		6:	IF (NOT(T_Station_Work.THWWorkStation.TAxisZ.T_CtrleSingle.xReset) AND (T_Station_Work.THWWorkStation.TAxisZ.T_CtrleSingle.xDone OR
			     T_Station_Work.THWWorkStation.TAxisZ.T_CtrleSingle.xErr)) OR
			    (NOT(T_Station_Work.THWWorkStation.TAxisS.T_CtrleSingle.xReset) AND (T_Station_Work.THWWorkStation.TAxisS.T_CtrleSingle.xDone OR
			     T_Station_Work.THWWorkStation.TAxisS.T_CtrleSingle.xErr)) THEN
				T_TwinSafe_Ctrle_Z_Axis.xError:=TRUE;	(* Resetten der Drive Optionskarte zu AX5000 Servo *)
				T_TwinSafe_Ctrle_S2_Axis.xError:=TRUE;	(* Resetten der Drive Optionskarte zu AX5000 Servo *)
				T_TwinSafe_Ctrle_S3_Axis.xError:=TRUE;	(* Resetten der Drive Optionskarte zu AX5000 Servo *)
				iStepResetHardware:=iStepResetHardware + 1;
			END_IF;
		7:	IF NOT(T_TwinSafe_Status_Z_Axis.xError) AND NOT(T_TwinSafe_Status_S2_Axis.xError) AND NOT(T_TwinSafe_Status_S3_Axis.xError) THEN
				T_TwinSafe_Ctrle_Z_Axis.xError:=FALSE;
				T_TwinSafe_Ctrle_S2_Axis.xError:=FALSE;
				T_TwinSafe_Ctrle_S3_Axis.xError:=FALSE;
				iStepResetHardware:=iStepResetHardware + 1;
			END_IF;
		8:	T_Station_Work.THWWorkStation.TAxisZ.T_CtrleSingle.xExecute:=TRUE;
			T_Station_Work.THWWorkStation.TAxisZ.T_CtrleSingle.iFunction:=1;	(* Resetten der NC Ebene *)
			T_Station_Work.THWWorkStation.TAxisS.T_CtrleSingle.xExecute:=TRUE;
			T_Station_Work.THWWorkStation.TAxisS.T_CtrleSingle.iFunction:=1;	(* Resetten der NC Ebene *)
			iStepResetHardware:=iStepResetHardware + 1;
		9:	IF (NOT(T_Station_Work.THWWorkStation.TAxisZ.T_CtrleSingle.xExecute) AND (T_Station_Work.THWWorkStation.TAxisZ.T_CtrleSingle.xDone
			OR T_Station_Work.THWWorkStation.TAxisZ.T_CtrleSingle.xErr))
			AND (NOT(T_Station_Work.THWWorkStation.TAxisS.T_CtrleSingle.xExecute) AND (T_Station_Work.THWWorkStation.TAxisS.T_CtrleSingle.xDone
			OR T_Station_Work.THWWorkStation.TAxisS.T_CtrleSingle.xErr)) THEN
				iStepResetHardware:=iStepResetHardware + 1;
			END_IF;
		10:	T_Station_Work.THWWorkStation.TAxisZ.T_CtrleSingle.xExecute:=TRUE;
			T_Station_Work.THWWorkStation.TAxisZ.T_CtrleSingle.iFunction:=27;	(* Resetten des AX5000 Servo *)
			T_Station_Work.THWWorkStation.TAxisS.T_CtrleSingle.xExecute:=(T_ExchgParam.bToolSpindleActive <> 1);		(* Nur ausführen wenn nicht Maxon Spindel aktiv ist *)
			T_Station_Work.THWWorkStation.TAxisS.T_CtrleSingle.iFunction:=27;	(* Resetten des AX5000 Servo *)
			iStepResetHardware:=iStepResetHardware + 1;
		11:	IF NOT(T_Station_Work.THWWorkStation.TAxisZ.T_CtrleSingle.xExecute) AND T_Station_Work.THWWorkStation.TAxisZ.T_CtrleSingle.xDone
			AND NOT(T_Station_Work.THWWorkStation.TAxisS.T_CtrleSingle.xExecute) AND T_Station_Work.THWWorkStation.TAxisS.T_CtrleSingle.xDone THEN
				T_Station_Work.THWWorkStation.TAxisZ.T_CtrleSingle.xExecute:=TRUE;
				T_Station_Work.THWWorkStation.TAxisZ.T_CtrleSingle.iFunction:=1;	(* Resetten der NC Ebene *)
				T_Station_Work.THWWorkStation.TAxisS.T_CtrleSingle.xExecute:=TRUE;
				T_Station_Work.THWWorkStation.TAxisS.T_CtrleSingle.iFunction:=1;	(* Resetten der NC Ebene *)
				iStepResetHardware:=iStepResetHardware + 1;
			END_IF;
		12:	IF NOT(T_Station_Work.THWWorkStation.TAxisZ.T_CtrleSingle.xExecute) AND T_Station_Work.THWWorkStation.TAxisZ.T_CtrleSingle.xDone
			OR NOT(T_Station_Work.THWWorkStation.TAxisS.T_CtrleSingle.xExecute) AND T_Station_Work.THWWorkStation.TAxisS.T_CtrleSingle.xDone THEN
				IF T_Station_Work.TControl.xResetHardwareActivateCurrent AND NOT(T_TwinSafe_Status_Z_Axis.xSTO) THEN
					T_Station_Work.THWWorkStation.TAxisZ.T_CtrleSingle.xExecute:=TRUE;
					T_Station_Work.THWWorkStation.TAxisZ.T_CtrleSingle.iFunction:=3;	(* Current ON *)
				END_IF;
				iStepResetHardware:=iStepResetHardware + 1;
			END_IF;
		13:	IF NOT(T_Station_Work.THWWorkStation.TAxisZ.T_CtrleSingle.xExecute) AND T_Station_Work.THWWorkStation.TAxisZ.T_CtrleSingle.xDone THEN
				iStepResetHardware:=1;
				IF NOT(xHardwareActive) THEN
					T_Station_Work.TControl.xActiveHardware:=FALSE;
				END_IF;
				T_Station_Work.TControl.xResetHardware:=FALSE;
			END_IF;
	END_CASE;
	TONWaitTimeOut(IN:=TRUE,PT:=T#3s);
	IF TONWaitTimeOut.Q THEN
		TONWaitTimeOut(IN:=FALSE);
		iStepResetHardware:=1;
		T_Station_Work.TControl.xResetHardware:=FALSE;
		T_Station_Work.THWWorkStation.TAxisZ.T_CtrleSingle.xReset:=TRUE;
		T_Station_Work.THWWorkStation.TAxisS.T_CtrleSingle.xReset:=TRUE;
		T_TwinSafe_Ctrle_Z_Axis.xError:=FALSE;
		T_TwinSafe_Ctrle_S2_Axis.xError:=FALSE;
		T_TwinSafe_Ctrle_S3_Axis.xError:=FALSE;
	END_IF;
ELSE
	TONWaitTimeOut(IN:=FALSE);
	iStepResetHardware:=1;
	T_Station_Work.TControl.xResetHardwareActivateCurrent:=FALSE;
END_IF;
IF T_Station_Work.TControl.xActiveHardware AND NOT(T_Station_Work.TControl.xResetHardware) THEN
	IF T_TwinSafe_Status_Z_Axis.xError OR ((T_TwinSafe_Status_S2_Axis.xError OR T_TwinSafe_Status_S3_Axis.xError) AND (T_ExchgParam.bToolSpindleActive <> 1)) THEN	(* Z Achse oder nur wenn nicht Maxon Spindel aktiv ist *)
		T_Station_Work.TControl.xResetHardware:=TRUE;
	END_IF;
END_IF;
xActiveHWStation:=T_Station_Work.TControl.xActiveHardware;
xActiveStation:=T_Station_Work.xActive;
RisingEdgeHWConfig(CLK:=xHardwareConfigError);
IF RisingEdgeHWConfig.Q THEN
	T_Station_Work.TControl.diErrorNr:=0;
	T_Station_Work.TControl.xError:=FALSE;
END_IF;

IF NOT(T_Station_Work.TControl.xActiveHardware) THEN
	T_Station_Work.TControl.xHWAxesActive:=TRUE;
	xHardwareConfigError:=FALSE;
	TONTickTime(IN:=FALSE);
	T_Station_Work.TControl.xActiveMovement:=FALSE;
	A01_AX5000_Parametrization;
	RETURN;
ELSE
	T_Station_Work.THWWorkStation.TAxisZ.T_DriveState:=stZDriveState;
	(* Zuweisung der Datenstrukturen der Aktuatoren als Pointer *)
	ptrTAxisZ:=ADR(T_Station_Work.THWWorkStation.TAxisZ);
	ptrTAxisS:=ADR(T_Station_Work.THWWorkStation.TAxisS);
	ptrTCylToolDeflection:=ADR(T_Station_Work.THWWorkStation.TCylToolDeflection);
	ptrTSensorTorque:=ADR(T_Station_Work.THWWorkStation.TSensorTorque);
	ptrTSensorTorqueOverload:=ADR(T_Station_Work.THWWorkStation.TSensorTorqueOverload);
	ptrTCylBrakeReleaseZAxis:=ADR(T_Station_Work.THWWorkStation.TCylBrakeReleaseZAxis);
	ptrTCylToolTorqueHC:=ADR(T_Station_Work.THWWorkStation.TCylToolTorqueHC);
	ptrTCylToolTorqueOverload:=ADR(T_Station_Work.THWWorkStation.TCylToolTorqueOverload);
	ptrTTorqueSensorMeasRange:=ADR(T_Station_Work.THWWorkStation.TTorqueSensorMeasRange);
	ptrTTorqueSensorControl:=ADR(T_Station_Work.THWWorkStation.TTorqueSensorControl);
	ptrTCylWorkpieceClamp:=ADR(T_Station_Work.THWWorkStation.TCylWorkpieceClamp);
	ptrTValveAirTable:=ADR(T_Station_Work.THWWorkStation.TValveAirTable);
	ptrTValveVacuumTable:=ADR(T_Station_Work.THWWorkStation.TValveVacuumTable);
	ptrTValveCleanNozzle:=ADR(T_Station_Work.THWWorkStation.TValveCleanNozzle);
	ptrTAxisBubbler:=ADR(T_Station_Work.THWWorkStation.TAxisBubbler);
	ptrTAxisFeedPump:=ADR(T_Station_Work.THWWorkStation.TAxisFeedPump);
	xEnableMasterModul:=TRUE;
	A01_DefineParameter;
	A01_InitParam;
END_IF;
(******************************************************************************************************************************************)
(****************************				         Check if Axis Active                                              *****************************)
(******************************************************************************************************************************************)
IF ptrTAxisZ^.T_CtrleSingle.xDone AND ptrTAxisS^.T_CtrleSingle.xDone THEN
	T_Station_Work.TControl.xHWAxesActive:=FALSE;
ELSE
	T_Station_Work.TControl.xHWAxesActive:=TRUE;
END_IF;
(******************************************************************************************************************************************)
(****************************	                        Check if Axis and Cylinder are Active                         *****************************)
(******************************************************************************************************************************************)
xCkeckAcitveMovement:=	(NOT(ptrTAxisZ^.T_CtrleSingle.xDone) AND NOT(ptrTAxisZ^.T_CtrleSingle.xErr))
						OR (NOT(ptrTAxisS^.T_CtrleSingle.xDone) AND NOT(ptrTAxisS^.T_CtrleSingle.xErr))
						OR (NOT(ptrTCylToolDeflection^.T_CtrleCyl.xDone) AND NOT(ptrTCylToolDeflection^.T_CtrleCyl.xErr))
						OR (NOT(ptrTCylToolTorqueHC^.T_CtrleCyl.xDone) AND NOT(ptrTCylToolTorqueHC^.T_CtrleCyl.xErr))
						OR (NOT(ptrTCylToolTorqueOverload^.T_CtrleCyl.xDone) AND NOT(ptrTCylToolTorqueOverload^.T_CtrleCyl.xErr))
						OR (NOT(ptrTTorqueSensorMeasRange^.T_CtrleCyl.xDone) AND NOT(ptrTTorqueSensorMeasRange^.T_CtrleCyl.xErr))
						OR (NOT(ptrTTorqueSensorControl^.T_CtrleCyl.xDone) AND NOT(ptrTTorqueSensorControl^.T_CtrleCyl.xErr))
						OR (NOT(ptrTCylBrakeReleaseZAxis^.T_CtrleCyl.xDone) AND NOT(ptrTCylBrakeReleaseZAxis^.T_CtrleCyl.xErr))
						OR (NOT(ptrTCylWorkpieceClamp^.T_CtrleCyl.xDone) AND NOT(ptrTCylWorkpieceClamp^.T_CtrleCyl.xErr))
						OR (NOT(ptrTValveAirTable^.T_CtrleCyl.xDone) AND NOT(ptrTValveAirTable^.T_CtrleCyl.xErr))
						OR (NOT(ptrTValveVacuumTable^.T_CtrleCyl.xDone) AND NOT(ptrTValveVacuumTable^.T_CtrleCyl.xErr))
						OR (NOT(ptrTValveCleanNozzle^.T_CtrleCyl.xDone) AND NOT(ptrTValveCleanNozzle^.T_CtrleCyl.xErr))
						OR (NOT(ptrTAxisBubbler^.T_CtrleDCAxis.xDone) AND NOT(ptrTAxisBubbler^.T_CtrleDCAxis.xErr))
						OR (NOT(ptrTAxisFeedPump^.T_CtrleDCAxis.xDone) AND NOT(ptrTAxisFeedPump^.T_CtrleDCAxis.xErr));
IF NOT(xCkeckAcitveMovement) THEN
	IF NOT(ptrTAxisZ^.T_CtrleSingle.xNotMoving) AND ptrTAxisZ^.T_CtrleSingle.xPower AND NOT(ptrTAxisZ^.T_CtrleSingle.xErr) THEN
		xCkeckAcitveMovement:=TRUE;
	END_IF;
	IF NOT(ptrTAxisS^.T_CtrleSingle.xNotMoving) AND ptrTAxisS^.T_CtrleSingle.xPower AND NOT(ptrTAxisS^.T_CtrleSingle.xErr) THEN
		xCkeckAcitveMovement:=TRUE;
	END_IF;
END_IF;
T_Station_Work.TControl.xActiveMovement:=xCkeckAcitveMovement;
(* HW Axis and Cylinder *)
HW_Axis_DC;	(* IGS3 *)
HW_AxisZ;
HW_AxisS;
HW_CylToolDeflection;
CASE T_ExchgParam.bToolSpindleActive OF
1:	(* Maxon Spindel *)
	HW_ToolTorqueHC;
	HW_ToolTorqueOverload;
	HW_TorqueSensor;
2,3:	(* Beckhoff Spindel *)
	HW_TorqueSensor2;
	HW_TorqueOverloadSensor;
END_CASE;
HW_TorqueSensorMeasureRange;
HW_TorqueSensorControl;
(* Beckhoff Spindel L = 0-2000(500)mNm	Beckhoff Spindel M = 0-500(100)mNm		-> nur Spindel M wird der kleine Bereich eingesetzt *)
IF (T_ExchgParam.bToolSpindleActive = 3) AND NOT(ptrTTorqueSensorMeasRange^.T_CtrleCyl.xExecute) AND ptrTTorqueSensorMeasRange^.T_CtrleCyl.xDone AND NOT(ptrTTorqueSensorMeasRange^.T_CtrleCyl.T_Standard.xActivOn) THEN
	ptrTTorqueSensorMeasRange^.T_CtrleCyl.iFunction:=2;
	ptrTTorqueSensorMeasRange^.T_CtrleCyl.xExecute:=TRUE;
END_IF;
HW_CylBrakeReleaseZAxis;
HW_CylWorkpieceClamp;
HW_ValveAirTable;
HW_ValveVacuumTable;
HW_ValveCleanNozzle; 	(* BEF *)
HW_TSensorToolSpindle_L_Connect;
(******************************************************************************************************************************************)
(****************************				                Reset Flags                                                           *****************************)
(******************************************************************************************************************************************)
ptrTAxisZ^.T_CtrleSingle.xReset:=FALSE;
ptrTAxisZ^.T_CtrleSingle.xExecute:=FALSE;
ptrTAxisS^.T_CtrleSingle.xReset:=FALSE;
ptrTAxisS^.T_CtrleSingle.xExecute:=FALSE;
ptrTCylToolDeflection^.T_CtrleCyl.xReset:=FALSE;
ptrTCylToolDeflection^.T_CtrleCyl.xExecute:=FALSE;
ptrTCylToolTorqueHC^.T_CtrleCyl.xReset:=FALSE;
ptrTCylToolTorqueHC^.T_CtrleCyl.xExecute:=FALSE;
ptrTCylToolTorqueOverload^.T_CtrleCyl.xReset:=FALSE;
ptrTCylToolTorqueOverload^.T_CtrleCyl.xExecute:=FALSE;
IF  (T_ExchgParam.bToolSpindleActive <> 1) THEN			(* diese Zylinder immer xDone schalten wenn nicht Maxon Spindel aktiv ist *)
	ptrTCylToolTorqueHC^.T_CtrleCyl.xDone:=TRUE;
	ptrTCylToolTorqueOverload^.T_CtrleCyl.xDone:=TRUE;
END_IF;
ptrTSensorTorque^.T_CtrleCyl.xReset:=FALSE;
ptrTSensorTorque^.T_CtrleCyl.xExecute:=FALSE;
ptrTSensorTorqueOverload^.T_CtrleCyl.xReset:=FALSE;
ptrTSensorTorqueOverload^.T_CtrleCyl.xExecute:=FALSE;
ptrTTorqueSensorMeasRange^.T_CtrleCyl.xReset:=FALSE;
ptrTTorqueSensorMeasRange^.T_CtrleCyl.xExecute:=FALSE;
ptrTTorqueSensorControl^.T_CtrleCyl.xReset:=FALSE;
ptrTTorqueSensorControl^.T_CtrleCyl.xExecute:=FALSE;
ptrTCylBrakeReleaseZAxis^.T_CtrleCyl.xReset:=FALSE;
ptrTCylBrakeReleaseZAxis^.T_CtrleCyl.xExecute:=FALSE;
ptrTCylWorkpieceClamp^.T_CtrleCyl.xReset:=FALSE;
ptrTCylWorkpieceClamp^.T_CtrleCyl.xExecute:=FALSE;
ptrTValveAirTable^.T_CtrleCyl.xReset:=FALSE;
ptrTValveAirTable^.T_CtrleCyl.xExecute:=FALSE;
ptrTValveVacuumTable^.T_CtrleCyl.xReset:=FALSE;
ptrTValveVacuumTable^.T_CtrleCyl.xExecute:=FALSE;
ptrTValveCleanNozzle^.T_CtrleCyl.xReset:=FALSE;
ptrTValveCleanNozzle^.T_CtrleCyl.xExecute:=FALSE;
ptrTAxisBubbler^.T_CtrleDCAxis.xReset:=FALSE;
ptrTAxisBubbler^.T_CtrleDCAxis.xExecute:=FALSE;
ptrTAxisFeedPump^.T_CtrleDCAxis.xReset:=FALSE;
ptrTAxisFeedPump^.T_CtrleDCAxis.xExecute:=FALSE;
END_FUNCTION_BLOCK
ACTION A01_AX5000_Parametrization:
IF T_ExchgParam.xWriteSoEParameter THEN
	CASE iStepWriteSoEParameter OF
	0:	CASE T_ExchgParam.bToolSpindleActive OF
		2:	iStepWriteSoEParameter:=iStepWriteSoEParameter + 1;
		3:	iStepWriteSoEParameter:=11;
		END_CASE;


	1:	fbGetAmsNetID(	sNetId:= '',
						iAxisId:= DWORD_TO_UINT(stS2RefIn.nAxisId),
						bExecute := TRUE);
		IF NOT fbGetAmsNetID.bBusy AND NOT fbGetAmsNetID.bError THEN
			fbGetAmsNetID.AxisNetId;
			sEtherCATNetId 	:= fbGetAmsNetID.AxisNetId;
			fbGetAmsNetID(	sNetId:= '',
							iAxisId:= DWORD_TO_UINT(stS2RefIn.nAxisId),
							bExecute := FALSE);
			iStepWriteSoEParameter:=iStepWriteSoEParameter + 1;
		ELSIF fbGetAmsNetID.bError THEN
			iStepWriteSoEParameter:=99;
		END_IF

	(* AX5000 in PreOP Mode setzen *)
	2:	fbSetSlaveState(	sNetId:= sEtherCATNetId,
						nSlaveAddr:= iSlaveAddr_AxisS,
						bExecute:= TRUE,
						tTimeout:= T#10s,
						reqState:= EC_DEVICE_STATE_PREOP);
		IF NOT(fbSetSlaveState.bBusy) OR fbSetSlaveState.bError THEN
			fbSetSlaveState(bExecute:=FALSE);
			iStepWriteSoEParameter:=iStepWriteSoEParameter + 1;
		END_IF;
	3:	fbGetSlaveState(	sNetId:=sEtherCATNetId,
						nSlaveAddr:=iSlaveAddr_AxisS,
						bExecute:=TRUE ,
						tTimeout:= t#10s,
						bBusy=> ,
						bError=> ,
						nErrId=> ,
						state=> );
		IF NOT fbGetSlaveState.bBusy AND NOT fbGetSlaveState.bError AND fbGetSlaveState.state.deviceState = fbSetSlaveState.reqState THEN
			fbGetSlaveState(bExecute:=FALSE);
			iStepWriteSoEParameter:=iStepWriteSoEParameter + 1;
		ELSIF fbGetSlaveState.bError THEN
			iStepWriteSoEParameter:=99;
		END_IF;

	(* P-0-0061 schreiben von Achse S2 *)
	4:	fbSoEWrite(	sNetId:=sEtherCATNetId,
					nSlaveAddr:= iSlaveAddr_AxisS,
					nIdn:=P_0_IDN + 61 ,
					nElement:=16#40 ,
					pSrcBuf:=ADR(T_Station_Parameter.T_AxisS2.uiP61) ,
					cbBufLen:=SIZEOF(T_Station_Parameter.T_AxisS2.uiP61) ,
					bExecute:=TRUE ,
					tTimeout:=t#10s ,
					nDriveNo:=0);		(* 0=Kanal A, 1=Kanal B *)
		IF NOT  fbSoEWrite.bBusy AND NOT fbSoEWrite.bError THEN
			fbSoEWrite(bExecute:=FALSE);
			iStepWriteSoEParameter:=iStepWriteSoEParameter + 1;
		ELSIF fbSoEWrite.bError THEN
			iStepWriteSoEParameter:=99;
		END_IF;

	(* P-0-0150 schreiben von Achse S2 *)
	5:	fbSoEWrite(	sNetId:=sEtherCATNetId,
					nSlaveAddr:= iSlaveAddr_AxisS,
					nIdn:=P_0_IDN + 150 ,
					nElement:=16#40 ,
					pSrcBuf:=ADR(T_Station_Parameter.T_AxisS2.bP150) ,
					cbBufLen:=SIZEOF(T_Station_Parameter.T_AxisS2.bP150) ,
					bExecute:=TRUE ,
					tTimeout:=t#10s ,
					nDriveNo:=0);		(* 0=Kanal A, 1=Kanal B *)
		IF NOT  fbSoEWrite.bBusy AND NOT fbSoEWrite.bError THEN
			fbSoEWrite(bExecute:=FALSE);
			iStepWriteSoEParameter:=iStepWriteSoEParameter + 1;
		ELSIF fbSoEWrite.bError THEN
			iStepWriteSoEParameter:=99;
		END_IF;

	(* AX5000 in OP Mode setzen *)
	6:	fbSetSlaveState(	sNetId:= sEtherCATNetId,
						nSlaveAddr:= iSlaveAddr_AxisS,
						bExecute:= TRUE,
						tTimeout:= T#10s,
						reqState:= EC_DEVICE_STATE_OP);
		IF NOT(fbSetSlaveState.bBusy) OR fbSetSlaveState.bError THEN
			fbSetSlaveState(bExecute:=FALSE);
			iStepWriteSoEParameter:=iStepWriteSoEParameter + 1;
		END_IF;
	7:	fbGetSlaveState(	sNetId:=sEtherCATNetId,
						nSlaveAddr:=iSlaveAddr_AxisS,
						bExecute:=TRUE ,
						tTimeout:= t#10s,
						bBusy=> ,
						bError=> ,
						nErrId=> ,
						state=> );
		IF NOT fbGetSlaveState.bBusy AND NOT fbGetSlaveState.bError AND (fbGetSlaveState.state.deviceState = fbSetSlaveState.reqState) THEN
			fbGetSlaveState(bExecute:=FALSE);
			T_ExchgParam.xWriteSoEParameter:=FALSE;
		ELSIF fbGetSlaveState.bError THEN
			iStepWriteSoEParameter:=99;
		ELSIF NOT fbGetSlaveState.bBusy AND NOT fbGetSlaveState.bError AND (fbGetSlaveState.state.deviceState = 82) THEN	(* deviceState = 82 => ERR_PREOP *)
			T_Station_Work.TControl.diErrorNr:=11;	(* Achsen MasterModul2 konnte den Spindelkopf L Kanal 1 nicht finden *)
			T_Station_Work.TControl.xError:=TRUE;
		END_IF;



	11:	fbGetAmsNetID(	sNetId:= '',
						iAxisId:= DWORD_TO_UINT(stS3RefIn.nAxisId),
						bExecute := TRUE);
		IF NOT fbGetAmsNetID.bBusy AND NOT fbGetAmsNetID.bError THEN
			fbGetAmsNetID.AxisNetId;
			sEtherCATNetId 	:= fbGetAmsNetID.AxisNetId;
			fbGetAmsNetID(	sNetId:= '',
							iAxisId:= DWORD_TO_UINT(stS3RefIn.nAxisId),
							bExecute := FALSE);
			iStepWriteSoEParameter:=iStepWriteSoEParameter + 1;
		ELSIF fbGetAmsNetID.bError THEN
			iStepWriteSoEParameter:=99;
		END_IF

	(* AX5000 in PreOP Mode setzen *)
	12:	fbSetSlaveState(	sNetId:= sEtherCATNetId,
						nSlaveAddr:= iSlaveAddr_AxisS,
						bExecute:= TRUE,
						tTimeout:= T#10s,
						reqState:= EC_DEVICE_STATE_PREOP);
		IF NOT(fbSetSlaveState.bBusy) OR fbSetSlaveState.bError THEN
			fbSetSlaveState(bExecute:=FALSE);
			iStepWriteSoEParameter:=iStepWriteSoEParameter + 1;
		END_IF;
	13:	fbGetSlaveState(	sNetId:=sEtherCATNetId,
						nSlaveAddr:=iSlaveAddr_AxisS,
						bExecute:=TRUE ,
						tTimeout:= t#10s,
						bBusy=> ,
						bError=> ,
						nErrId=> ,
						state=> );
		IF NOT fbGetSlaveState.bBusy AND NOT fbGetSlaveState.bError AND fbGetSlaveState.state.deviceState = fbSetSlaveState.reqState THEN
			fbGetSlaveState(bExecute:=FALSE);
			iStepWriteSoEParameter:=iStepWriteSoEParameter + 1;
		ELSIF fbGetSlaveState.bError THEN
			iStepWriteSoEParameter:=99;
		END_IF;

	(* P-0-0061 schreiben von Achse S3 *)
	14:	fbSoEWrite(	sNetId:=sEtherCATNetId,
					nSlaveAddr:= iSlaveAddr_AxisS,
					nIdn:=P_0_IDN + 61 ,
					nElement:=16#40 ,
					pSrcBuf:=ADR(T_Station_Parameter.T_AxisS3.uiP61) ,
					cbBufLen:=SIZEOF(T_Station_Parameter.T_AxisS3.uiP61) ,
					bExecute:=TRUE ,
					tTimeout:=t#10s ,
					nDriveNo:=1);		(* 0=Kanal A, 1=Kanal B *)
		IF NOT  fbSoEWrite.bBusy AND NOT fbSoEWrite.bError THEN
			fbSoEWrite(bExecute:=FALSE);
			iStepWriteSoEParameter:=iStepWriteSoEParameter + 1;
		ELSIF fbSoEWrite.bError THEN
			iStepWriteSoEParameter:=99;
		END_IF;

	(* P-0-0150 schreiben von Achse S2 *)
	15:	fbSoEWrite(	sNetId:=sEtherCATNetId,
					nSlaveAddr:= iSlaveAddr_AxisS,
					nIdn:=P_0_IDN + 150 ,
					nElement:=16#40 ,
					pSrcBuf:=ADR(T_Station_Parameter.T_AxisS3.bP150) ,
					cbBufLen:=SIZEOF(T_Station_Parameter.T_AxisS3.bP150) ,
					bExecute:=TRUE ,
					tTimeout:=t#10s ,
					nDriveNo:=1);		(* 0=Kanal A, 1=Kanal B *)
		IF NOT  fbSoEWrite.bBusy AND NOT fbSoEWrite.bError THEN
			fbSoEWrite(bExecute:=FALSE);
			iStepWriteSoEParameter:=iStepWriteSoEParameter + 1;
		ELSIF fbSoEWrite.bError THEN
			iStepWriteSoEParameter:=99;
		END_IF;

	(* AX5000 in OP Mode setzen *)
	16:	fbSetSlaveState(	sNetId:= sEtherCATNetId,
						nSlaveAddr:= iSlaveAddr_AxisS,
						bExecute:= TRUE,
						tTimeout:= T#10s,
						reqState:= EC_DEVICE_STATE_OP);
		IF NOT(fbSetSlaveState.bBusy) OR fbSetSlaveState.bError THEN
			fbSetSlaveState(bExecute:=FALSE);
			iStepWriteSoEParameter:=iStepWriteSoEParameter + 1;
		END_IF;
	17:	fbGetSlaveState(	sNetId:=sEtherCATNetId,
						nSlaveAddr:=iSlaveAddr_AxisS,
						bExecute:=TRUE ,
						tTimeout:= t#10s,
						bBusy=> ,
						bError=> ,
						nErrId=> ,
						state=> );
		IF NOT fbGetSlaveState.bBusy AND NOT fbGetSlaveState.bError AND (fbGetSlaveState.state.deviceState = fbSetSlaveState.reqState) THEN
			fbGetSlaveState(bExecute:=FALSE);
			T_ExchgParam.xWriteSoEParameter:=FALSE;
		ELSIF fbGetSlaveState.bError THEN
			iStepWriteSoEParameter:=99;
		ELSIF NOT fbGetSlaveState.bBusy AND NOT fbGetSlaveState.bError AND (fbGetSlaveState.state.deviceState = 82) THEN	(* deviceState = 82 => ERR_PREOP *)
			T_Station_Work.TControl.diErrorNr:=12;	(* Achsen MasterModul2 konnte den Spindelkopf M Kanal 2 nicht finden *)
			T_Station_Work.TControl.xError:=TRUE;
		END_IF;
	ELSE

		fbGetAmsNetID(bExecute:=FALSE);
		fbSetSlaveState(bExecute:=FALSE);
		fbGetSlaveState(bExecute:=FALSE);
		fbSoEWrite(bExecute:=FALSE);
		iStepWriteSoEParameter:=0;
		T_Station_Work.TControl.diErrorNr:=10;	(* AX5000 Parameter konnte nicht erfolgreich geschrieben werden *)
		T_Station_Work.TControl.xError:=TRUE;

	END_CASE
ELSE
	iStepWriteSoEParameter:=0;
END_IF



IF xReadSoEParameter THEN
	CASE iStepReadSoEParameter OF
	0:	fbGetAmsNetID(	sNetId:= '',
						iAxisId:= DWORD_TO_UINT(stS2RefIn.nAxisId),
						bExecute := TRUE);
		IF NOT fbGetAmsNetID.bBusy AND NOT fbGetAmsNetID.bError THEN
			fbGetAmsNetID.AxisNetId;
			sEtherCATNetId 	:= fbGetAmsNetID.AxisNetId;
			fbGetAmsNetID(	sNetId:= '',
							iAxisId:= DWORD_TO_UINT(stS2RefIn.nAxisId),
							bExecute := FALSE);
			iStepReadSoEParameter:=iStepReadSoEParameter + 1;
		END_IF

	(* P-0-0061 lesen von Achse S2 *)
	1:	fbSoERead(	sNetId:=sEtherCATNetId,
					nSlaveAddr:= iSlaveAddr_AxisS,
					nIdn:=P_0_IDN + 61 ,
					nElement:=16#40 ,
					pDstBuf:=ADR(T_Station_Parameter.T_AxisS2.uiP61) ,
					cbBufLen:=SIZEOF(T_Station_Parameter.T_AxisS2.uiP61) ,
					bExecute:=TRUE ,
					tTimeout:=t#10s ,
					nDriveNo:=0);		(* 0=Kanal A, 1=Kanal B *)
		IF NOT  fbSoERead.bBusy AND NOT fbSoERead.bError THEN
			FBSoERead(bExecute:=FALSE);
			iStepReadSoEParameter:=iStepReadSoEParameter + 1;
		ELSIF fbSoERead.bError THEN
			;
		END_IF;

	(* P-0-0150 lesen von Achse S2 *)
	2:	fbSoERead(	sNetId:=sEtherCATNetId,
					nSlaveAddr:= iSlaveAddr_AxisS,
					nIdn:=P_0_IDN + 150 ,
					nElement:=16#40 ,
					pDstBuf:=ADR(T_Station_Parameter.T_AxisS2.bP150) ,
					cbBufLen:=SIZEOF(T_Station_Parameter.T_AxisS2.bP150) ,
					bExecute:=TRUE ,
					tTimeout:=t#10s ,
					nDriveNo:=0);		(* 0=Kanal A, 1=Kanal B *)
		IF NOT  fbSoERead.bBusy AND NOT fbSoERead.bError THEN
			FBSoERead(bExecute:=FALSE);
			iStepReadSoEParameter:=10;
		ELSIF fbSoERead.bError THEN
			;
		END_IF;

	10:	fbGetAmsNetID(	sNetId:= '',
						iAxisId:= DWORD_TO_UINT(stS3RefIn.nAxisId),
						bExecute := TRUE);
		IF NOT fbGetAmsNetID.bBusy AND NOT fbGetAmsNetID.bError THEN
			fbGetAmsNetID.AxisNetId;
			sEtherCATNetId 	:= fbGetAmsNetID.AxisNetId;
			fbGetAmsNetID(	sNetId:= '',
							iAxisId:= DWORD_TO_UINT(stS3RefIn.nAxisId),
							bExecute := FALSE);
			iStepReadSoEParameter:=iStepReadSoEParameter + 1;
		END_IF

	(* P-0-0061 lesen von Achse S3 *)
	11:	fbSoERead(	sNetId:=sEtherCATNetId,
					nSlaveAddr:= iSlaveAddr_AxisS,
					nIdn:=P_0_IDN + 61 ,
					nElement:=16#40 ,
					pDstBuf:=ADR(T_Station_Parameter.T_AxisS3.uiP61) ,
					cbBufLen:=SIZEOF(T_Station_Parameter.T_AxisS3.uiP61) ,
					bExecute:=TRUE ,
					tTimeout:=t#10s ,
					nDriveNo:=1);		(* 0=Kanal A, 1=Kanal B *)
		IF NOT  fbSoERead.bBusy AND NOT fbSoERead.bError THEN
			FBSoERead(bExecute:=FALSE);
			iStepReadSoEParameter:=iStepReadSoEParameter + 1;
		ELSIF fbSoERead.bError THEN
			;
		END_IF;

	(* P-0-0150 lesen von Achse S3 *)
	12:	fbSoERead(	sNetId:=sEtherCATNetId,
					nSlaveAddr:= iSlaveAddr_AxisS,
					nIdn:=P_0_IDN + 150 ,
					nElement:=16#40 ,
					pDstBuf:=ADR(T_Station_Parameter.T_AxisS3.bP150) ,
					cbBufLen:=SIZEOF(T_Station_Parameter.T_AxisS3.bP150) ,
					bExecute:=TRUE ,
					tTimeout:=t#10s ,
					nDriveNo:=1);		(* 0=Kanal A, 1=Kanal B *)
		IF NOT  fbSoERead.bBusy AND NOT fbSoERead.bError THEN
			FBSoERead(bExecute:=FALSE);
			xReadSoEParameter:=FALSE;
		ELSIF fbSoERead.bError THEN
			;
		END_IF;
	END_CASE
ELSE
	iStepReadSoEParameter:=0;
END_IF
END_ACTION
ACTION A01_DefineParameter:
(*Define Constant Axis Param Working Station*)
	gcarAxisConfig[gciAxisZ_St1].rIncFast				:=T_ExchgParam.T_TeachIn.arTeachSelStep[gciAxisZ_St1];
	gcarAxisConfig[gciAxisZ_St1].rIncSlow			:=T_ExchgParam.T_TeachIn.arTeachSelStep[gciAxisZ_St1];
	gcarAxisConfig[gciAxisZ_St1].rPositionSpeed		:=30.0;
	gcarAxisConfig[gciAxisZ_St1].rRefPosition			:=T_Station_Parameter.T_AxisState.rPositionReferenceZAxis;
	gcarAxisConfig[gciAxisZ_St1].rRefSpeed			:=20.0;
	gcarAxisConfig[gciAxisZ_St1].rVelFast				:=T_ExchgParam.T_TeachIn.arTeachSelVel[gciAxisZ_St1];
	gcarAxisConfig[gciAxisZ_St1].rVelSlow			:=T_ExchgParam.T_TeachIn.arTeachSelVel[gciAxisZ_St1];
	gcarAxisConfig[gciAxisZ_St1].rAcceleration		:=80000.0;	(* 88000 *)
	gcarAxisConfig[gciAxisZ_St1].rDeceleration		:=80000.0;	(* 88000 *)
	gcarAxisConfig[gciAxisZ_St1].rJerk				:=30000.0;	(* 88000 *)
	ptrTAxisZ^.T_Config_Gen.wPosLimitSwitchBit	:=8;
	ptrTAxisZ^.T_Config_Gen.wNegLimitSwitchBit	:=16;

	gcarAxisConfig[gciAxisS_St1].rIncFast				:=T_ExchgParam.T_TeachIn.arTeachSelStep[gciAxisS_St1];
	gcarAxisConfig[gciAxisS_St1].rIncSlow			:=T_ExchgParam.T_TeachIn.arTeachSelStep[gciAxisS_St1];
	gcarAxisConfig[gciAxisS_St1].rPositionSpeed		:=0.0;
	gcarAxisConfig[gciAxisS_St1].rRefPosition			:=0.0;
	gcarAxisConfig[gciAxisS_St1].rRefSpeed			:=0.0;
	gcarAxisConfig[gciAxisS_St1].rVelFast				:=T_ExchgParam.T_TeachIn.arTeachSelVel[gciAxisS_St1];
	gcarAxisConfig[gciAxisS_St1].rVelSlow			:=T_ExchgParam.T_TeachIn.arTeachSelVel[gciAxisS_St1];
	gcarAxisConfig[gciAxisS_St1].rAcceleration		:=200000.0;
	gcarAxisConfig[gciAxisS_St1].rDeceleration		:=200000.0;
	gcarAxisConfig[gciAxisS_St1].rJerk				:=200000.0;
	CASE T_ExchgParam.bToolSpindleActive OF
	1:	(* Maxon Spindel *)
		T_Station_Work.THWWorkStation.TCtrlWork.rMaxToolSpindleSpeed:=grMaxSAxis_Speed_SM * T_Station_Parameter.T_TorqueSystem.rGearRatioGearBox;
	2:	(* Beckhoff Spindel L *)
		T_Station_Work.THWWorkStation.TCtrlWork.rMaxToolSpindleSpeed:=grMaxSAxis_Speed_L;
	3:	(* Beckhoff Spindel M *)
		T_Station_Work.THWWorkStation.TCtrlWork.rMaxToolSpindleSpeed:=grMaxSAxis_Speed_M;
	END_CASE;
END_ACTION
ACTION A01_InitParam:
(* Axis Z *)
ptrTAxisZ^.T_Config_Gen.iTyp													:=1;
ptrTAxisZ^.T_Config_Setting.xSoftwareLimitNeg									:=FALSE;
ptrTAxisZ^.T_Config_Setting.xSoftwareLimitPos									:=FALSE;
ptrTAxisZ^.T_Config_Setting.xHardwareLimitNeg									:=TRUE;
ptrTAxisZ^.T_Config_Setting.xHardwareLimitPos									:=TRUE;
ptrTAxisZ^.T_CtrleSingle.xMoveAwayFromHWLimitSwitchActive						:=TRUE;
ptrTAxisZ^.T_CtrleSingle.xAX5000Active											:=TRUE;
ptrTAxisZ^.T_Config_Setting.xAbsoluteEncoder									:=TRUE;
ptrTAxisZ^.T_CtrleSingle.xKL2541Active											:=FALSE;
ptrTAxisZ^.T_CtrleSingle.lrAcceleration											:=gcarAxisConfig[gciAxisZ_St1].rAcceleration;
ptrTAxisZ^.T_CtrleSingle.lrDecceleration											:=gcarAxisConfig[gciAxisZ_St1].rDeceleration;
ptrTAxisZ^.T_CtrleSingle.lrJerk													:=gcarAxisConfig[gciAxisZ_St1].rJerk;

(* Axis S *)
ptrTAxisS^.T_Config_Gen.iTyp													:=2;
ptrTAxisS^.T_Config_Setting.xSoftwareLimitNeg									:=FALSE;
ptrTAxisS^.T_Config_Setting.xSoftwareLimitPos									:=FALSE;
ptrTAxisS^.T_Config_Setting.xHardwareLimitNeg									:=FALSE;
ptrTAxisS^.T_Config_Setting.xHardwareLimitPos									:=FALSE;
ptrTAxisS^.T_CtrleSingle.xMoveAwayFromHWLimitSwitchActive						:=FALSE;
ptrTAxisS^.T_CtrleSingle.xAX5000Active											:=FALSE;
ptrTAxisS^.T_Config_Setting.xAbsoluteEncoder									:=FALSE;
ptrTAxisS^.T_CtrleSingle.xKL2541Active											:=FALSE;
ptrTAxisS^.T_CtrleSingle.lrAcceleration											:=gcarAxisConfig[gciAxisS_St1].rAcceleration;
ptrTAxisS^.T_CtrleSingle.lrDecceleration											:=gcarAxisConfig[gciAxisS_St1].rDeceleration;
ptrTAxisS^.T_CtrleSingle.lrJerk													:=gcarAxisConfig[gciAxisS_St1].rJerk;

(* Config Cyl ToolDeflection *)
ptrTCylToolDeflection^.iCylinderTpye											:=1;
ptrTCylToolDeflection^.T_CtrleCyl.xFBActiv										:=T_Station_Work.TControl.xEnable;
ptrTCylToolDeflection^.T_Config.xActivState										:=TRUE;
ptrTCylToolDeflection^.T_Config.xCtrlePosOff										:=FALSE;
ptrTCylToolDeflection^.T_Config.xCtrlePosOn										:=FALSE;
ptrTCylToolDeflection^.T_Config.tTimeOut										:=T#0s;
ptrTCylToolDeflection^.T_Config.tDelayOff										:=ptrTCylToolDeflection^.T_Config.tDelayOff;
ptrTCylToolDeflection^.T_Config.tDelayOn										:=ptrTCylToolDeflection^.T_Config.tDelayOn;
ptrTCylToolDeflection^.T_CtrleCyl.T_Standard.tDelayAfterSensorOff					:=ptrTCylToolDeflection^.T_CtrleCyl.T_Standard.tDelayAfterSensorOff;
ptrTCylToolDeflection^.T_CtrleCyl.T_Standard.tDelayAfterSensorOn					:=ptrTCylToolDeflection^.T_CtrleCyl.T_Standard.tDelayAfterSensorOn;
ptrTCylToolDeflection^.T_CtrleCyl.T_Standard.tDelayActiv							:=T#0s;
ptrTCylToolDeflection^.T_Config.tDelayPreOff										:=T#0s;
ptrTCylToolDeflection^.T_Config.tDelayPreOn										:=T#0s;

(* Config Cyl ToolTorqueHC *)
ptrTCylToolTorqueHC^.iCylinderTpye											:=2;
ptrTCylToolTorqueHC^.T_CtrleCyl.xFBActiv										:=T_Station_Work.TControl.xEnable;
ptrTCylToolTorqueHC^.T_Config.xActivState										:=TRUE;
ptrTCylToolTorqueHC^.T_Config.xCtrlePosOff										:=FALSE;
ptrTCylToolTorqueHC^.T_Config.xCtrlePosOn										:=FALSE;
ptrTCylToolTorqueHC^.T_Config.tTimeOut										:=T#0s;
ptrTCylToolTorqueHC^.T_Config.tDelayOff										:=ptrTCylToolTorqueHC^.T_Config.tDelayOff;
ptrTCylToolTorqueHC^.T_Config.tDelayOn										:=ptrTCylToolTorqueHC^.T_Config.tDelayOn;
ptrTCylToolTorqueHC^.T_CtrleCyl.T_Standard.tDelayAfterSensorOff					:=ptrTCylToolTorqueHC^.T_CtrleCyl.T_Standard.tDelayAfterSensorOff;
ptrTCylToolTorqueHC^.T_CtrleCyl.T_Standard.tDelayAfterSensorOn					:=ptrTCylToolTorqueHC^.T_CtrleCyl.T_Standard.tDelayAfterSensorOn;
ptrTCylToolTorqueHC^.T_CtrleCyl.T_Standard.tDelayActiv							:=T#0s;
ptrTCylToolTorqueHC^.T_Config.tDelayPreOff										:=T#0s;
ptrTCylToolTorqueHC^.T_Config.tDelayPreOn										:=T#0s;

(* Config Cyl ToolTorqueOverload *)
ptrTCylToolTorqueOverload^.iCylinderTpye										:=3;
ptrTCylToolTorqueOverload^.T_CtrleCyl.xFBActiv									:=T_Station_Work.TControl.xEnable;
ptrTCylToolTorqueOverload^.T_Config.xActivState									:=TRUE;
ptrTCylToolTorqueOverload^.T_Config.xCtrlePosOff								:=FALSE;
ptrTCylToolTorqueOverload^.T_Config.xCtrlePosOn								:=FALSE;
ptrTCylToolTorqueOverload^.T_Config.tTimeOut									:=T#0s;
ptrTCylToolTorqueOverload^.T_Config.tDelayOff									:=ptrTCylToolTorqueOverload^.T_Config.tDelayOff;
ptrTCylToolTorqueOverload^.T_Config.tDelayOn									:=ptrTCylToolTorqueOverload^.T_Config.tDelayOn;
ptrTCylToolTorqueOverload^.T_CtrleCyl.T_Standard.tDelayAfterSensorOff				:=ptrTCylToolTorqueOverload^.T_CtrleCyl.T_Standard.tDelayAfterSensorOff;
ptrTCylToolTorqueOverload^.T_CtrleCyl.T_Standard.tDelayAfterSensorOn				:=ptrTCylToolTorqueOverload^.T_CtrleCyl.T_Standard.tDelayAfterSensorOn;
ptrTCylToolTorqueOverload^.T_CtrleCyl.T_Standard.tDelayActiv						:=T#0s;
ptrTCylToolTorqueOverload^.T_Config.tDelayPreOff								:=T#0s;
ptrTCylToolTorqueOverload^.T_Config.tDelayPreOn								:=T#0s;

(* Config Cyl BrakeReleaseZAxis *)
ptrTCylBrakeReleaseZAxis^.iCylinderTpye										:=4;
ptrTCylBrakeReleaseZAxis^.T_CtrleCyl.xFBActiv									:=T_Station_Work.TControl.xEnable;
ptrTCylBrakeReleaseZAxis^.T_Config.xActivState									:=TRUE;
ptrTCylBrakeReleaseZAxis^.T_Config.xCtrlePosOff									:=FALSE;
ptrTCylBrakeReleaseZAxis^.T_Config.xCtrlePosOn									:=FALSE;
ptrTCylBrakeReleaseZAxis^.T_Config.tTimeOut									:=REAL_TO_TIME(T_Station_Parameter.TCylBrakeReleaseZAxis.rTimeOutError * 1000.0);
ptrTCylBrakeReleaseZAxis^.T_Config.tDelayOff									:=REAL_TO_TIME(T_Station_Parameter.TCylBrakeReleaseZAxis.rTimeDelayOFF * 1000.0);
ptrTCylBrakeReleaseZAxis^.T_Config.tDelayOn									:=REAL_TO_TIME(T_Station_Parameter.TCylBrakeReleaseZAxis.rTimeDelayON * 1000.0);
ptrTCylBrakeReleaseZAxis^.T_CtrleCyl.T_Standard.tDelayAfterSensorOff				:=REAL_TO_TIME(T_Station_Parameter.TCylBrakeReleaseZAxis.rTimeAfterSensorOFF * 1000.0);
ptrTCylBrakeReleaseZAxis^.T_CtrleCyl.T_Standard.tDelayAfterSensorOn				:=REAL_TO_TIME(T_Station_Parameter.TCylBrakeReleaseZAxis.rTimeAfterSensorON * 1000.0);
ptrTCylBrakeReleaseZAxis^.T_CtrleCyl.T_Standard.tDelayActiv						:=T#0s;
ptrTCylBrakeReleaseZAxis^.T_Config.tDelayPreOff									:=T#0s;
ptrTCylBrakeReleaseZAxis^.T_Config.tDelayPreOn								:=T#0s;

(* Config Cyl WorkpieceClamp *)
ptrTCylWorkpieceClamp^.iCylinderTpye											:=5;
ptrTCylWorkpieceClamp^.T_CtrleCyl.xFBActiv										:=T_Station_Work.TControl.xEnable;
ptrTCylWorkpieceClamp^.T_Config.xActivState									:=TRUE;
ptrTCylWorkpieceClamp^.T_Config.xCtrlePosOff									:=FALSE;
ptrTCylWorkpieceClamp^.T_Config.xCtrlePosOn									:=FALSE;
ptrTCylWorkpieceClamp^.T_Config.tTimeOut										:=ptrTCylWorkpieceClamp^.T_Config.tTimeOut;
ptrTCylWorkpieceClamp^.T_Config.tDelayOff										:=ptrTCylWorkpieceClamp^.T_Config.tDelayOff;
ptrTCylWorkpieceClamp^.T_Config.tDelayOn										:=ptrTCylWorkpieceClamp^.T_Config.tDelayOn;
ptrTCylWorkpieceClamp^.T_CtrleCyl.T_Standard.tDelayAfterSensorOff				:=ptrTCylWorkpieceClamp^.T_CtrleCyl.T_Standard.tDelayAfterSensorOff;
ptrTCylWorkpieceClamp^.T_CtrleCyl.T_Standard.tDelayAfterSensorOn				:=ptrTCylWorkpieceClamp^.T_CtrleCyl.T_Standard.tDelayAfterSensorOn;
ptrTCylWorkpieceClamp^.T_CtrleCyl.T_Standard.tDelayActiv						:=T#0s;
ptrTCylWorkpieceClamp^.T_Config.tDelayPreOff									:=T#0s;
ptrTCylWorkpieceClamp^.T_Config.tDelayPreOn									:=T#0s;

(* Config Valve AirTable *)
ptrTValveAirTable^.iCylinderTpye												:=6;
ptrTValveAirTable^.T_CtrleCyl.xFBActiv											:=T_Station_Work.TControl.xEnable;
ptrTValveAirTable^.T_Config.xActivState											:=TRUE;
ptrTValveAirTable^.T_Config.xCtrlePosOff											:=FALSE;
ptrTValveAirTable^.T_Config.xCtrlePosOn										:=FALSE;
ptrTValveAirTable^.T_Config.tTimeOut											:=ptrTValveAirTable^.T_Config.tTimeOut;
ptrTValveAirTable^.T_Config.tDelayOff											:=ptrTValveAirTable^.T_Config.tDelayOff;
ptrTValveAirTable^.T_Config.tDelayOn											:=ptrTValveAirTable^.T_Config.tDelayOn;
ptrTValveAirTable^.T_CtrleCyl.T_Standard.tDelayAfterSensorOff						:=ptrTValveAirTable^.T_CtrleCyl.T_Standard.tDelayAfterSensorOff;
ptrTValveAirTable^.T_CtrleCyl.T_Standard.tDelayAfterSensorOn						:=ptrTValveAirTable^.T_CtrleCyl.T_Standard.tDelayAfterSensorOn;
ptrTValveAirTable^.T_CtrleCyl.T_Standard.tDelayActiv								:=T#0s;
ptrTValveAirTable^.T_Config.tDelayPreOff										:=T#0s;
ptrTValveAirTable^.T_Config.tDelayPreOn										:=T#0s;

(* Config Valve VacuumTable *)
ptrTValveVacuumTable^.iCylinderTpye											:=7;
ptrTValveVacuumTable^.T_CtrleCyl.xFBActiv										:=T_Station_Work.TControl.xEnable;
ptrTValveVacuumTable^.T_Config.xActivState										:=TRUE;
ptrTValveVacuumTable^.T_Config.xCtrlePosOff									:=FALSE;
ptrTValveVacuumTable^.T_Config.xCtrlePosOn									:=FALSE;
ptrTValveVacuumTable^.T_Config.tTimeOut										:=ptrTValveVacuumTable^.T_Config.tTimeOut;
ptrTValveVacuumTable^.T_Config.tDelayOff										:=ptrTValveVacuumTable^.T_Config.tDelayOff;
ptrTValveVacuumTable^.T_Config.tDelayOn										:=ptrTValveVacuumTable^.T_Config.tDelayOn;
ptrTValveVacuumTable^.T_CtrleCyl.T_Standard.tDelayAfterSensorOff					:=ptrTValveVacuumTable^.T_CtrleCyl.T_Standard.tDelayAfterSensorOff;
ptrTValveVacuumTable^.T_CtrleCyl.T_Standard.tDelayAfterSensorOn					:=ptrTValveVacuumTable^.T_CtrleCyl.T_Standard.tDelayAfterSensorOn;
ptrTValveVacuumTable^.T_CtrleCyl.T_Standard.tDelayActiv							:=T#0s;
ptrTValveVacuumTable^.T_Config.tDelayPreOff									:=T#0s;
ptrTValveVacuumTable^.T_Config.tDelayPreOn									:=T#0s;

(* Config Valve Cleaning nozzle  *)
ptrTValveCleanNozzle^.iCylinderTpye											:=8;
ptrTValveCleanNozzle^.T_CtrleCyl.xFBActiv										:=T_Station_Work.TControl.xEnable;
ptrTValveCleanNozzle^.T_Config.xActivState										:=TRUE;
ptrTValveCleanNozzle^.T_Config.xCtrlePosOff										:=FALSE;
ptrTValveCleanNozzle^.T_Config.xCtrlePosOn										:=FALSE;
ptrTValveCleanNozzle^.T_Config.tTimeOut										:=ptrTValveCleanNozzle^.T_Config.tTimeOut;
ptrTValveCleanNozzle^.T_Config.tDelayOff										:=ptrTValveCleanNozzle^.T_Config.tDelayOff;
ptrTValveCleanNozzle^.T_Config.tDelayOn										:=ptrTValveCleanNozzle^.T_Config.tDelayOn;
ptrTValveCleanNozzle^.T_CtrleCyl.T_Standard.tDelayAfterSensorOff					:=ptrTValveCleanNozzle^.T_CtrleCyl.T_Standard.tDelayAfterSensorOff;
ptrTValveCleanNozzle^.T_CtrleCyl.T_Standard.tDelayAfterSensorOn					:=ptrTValveCleanNozzle^.T_CtrleCyl.T_Standard.tDelayAfterSensorOn;
ptrTValveCleanNozzle^.T_CtrleCyl.T_Standard.tDelayActiv							:=T#0s;
ptrTValveCleanNozzle^.T_Config.tDelayPreOff										:=T#0s;
ptrTValveCleanNozzle^.T_Config.tDelayPreOn										:=T#0s;

(* Config SensorTorque *)
ptrTSensorTorque^.iCylinderTpye												:=20;
ptrTSensorTorque^.T_CtrleCyl.xFBActiv											:=T_Station_Work.TControl.xEnable;
ptrTSensorTorque^.T_Config.xActivState											:=TRUE;
ptrTSensorTorque^.T_Config.xCtrlePosOff											:=FALSE;
ptrTSensorTorque^.T_Config.xCtrlePosOn										:=FALSE;
ptrTSensorTorque^.T_Config.tTimeOut											:=T#0s;
ptrTSensorTorque^.T_Config.tDelayOff											:=ptrTSensorTorque^.T_Config.tDelayOff;
ptrTSensorTorque^.T_Config.tDelayOn											:=ptrTSensorTorque^.T_Config.tDelayOn;
ptrTSensorTorque^.T_CtrleCyl.T_Standard.tDelayAfterSensorOff						:=ptrTSensorTorque^.T_CtrleCyl.T_Standard.tDelayAfterSensorOff;
ptrTSensorTorque^.T_CtrleCyl.T_Standard.tDelayAfterSensorOn						:=ptrTSensorTorque^.T_CtrleCyl.T_Standard.tDelayAfterSensorOn;
ptrTSensorTorque^.T_CtrleCyl.T_Standard.tDelayActiv								:=T#0s;
ptrTSensorTorque^.T_Config.tDelayPreOff										:=T#0s;
ptrTSensorTorque^.T_Config.tDelayPreOn										:=T#0s;

(* Config SensorTorqueOverload *)
ptrTSensorTorqueOverload^.iCylinderTpye										:=21;
ptrTSensorTorqueOverload^.T_CtrleCyl.xFBActiv									:=T_Station_Work.TControl.xEnable;
ptrTSensorTorqueOverload^.T_Config.xActivState									:=TRUE;
ptrTSensorTorqueOverload^.T_Config.xCtrlePosOff									:=FALSE;
ptrTSensorTorqueOverload^.T_Config.xCtrlePosOn								:=FALSE;
ptrTSensorTorqueOverload^.T_Config.tTimeOut									:=T#0s;
ptrTSensorTorqueOverload^.T_Config.tDelayOff									:=ptrTSensorTorqueOverload^.T_Config.tDelayOff;
ptrTSensorTorqueOverload^.T_Config.tDelayOn									:=ptrTSensorTorqueOverload^.T_Config.tDelayOn;
ptrTSensorTorqueOverload^.T_CtrleCyl.T_Standard.tDelayAfterSensorOff				:=ptrTSensorTorqueOverload^.T_CtrleCyl.T_Standard.tDelayAfterSensorOff;
ptrTSensorTorqueOverload^.T_CtrleCyl.T_Standard.tDelayAfterSensorOn				:=ptrTSensorTorqueOverload^.T_CtrleCyl.T_Standard.tDelayAfterSensorOn;
ptrTSensorTorqueOverload^.T_CtrleCyl.T_Standard.tDelayActiv						:=T#0s;
ptrTSensorTorqueOverload^.T_Config.tDelayPreOff								:=T#0s;
ptrTSensorTorqueOverload^.T_Config.tDelayPreOn								:=T#0s;

(* Config Sensor TorqueSensorMeasRange *)
ptrTTorqueSensorMeasRange^.iCylinderTpye									:=22;
ptrTTorqueSensorMeasRange^.T_CtrleCyl.xFBActiv								:=T_Station_Work.TControl.xEnable;
ptrTTorqueSensorMeasRange^.T_Config.xActivState								:=TRUE;
ptrTTorqueSensorMeasRange^.T_Config.xCtrlePosOff								:=FALSE;
ptrTTorqueSensorMeasRange^.T_Config.xCtrlePosOn								:=FALSE;
ptrTTorqueSensorMeasRange^.T_Config.tTimeOut									:=T#0s;
ptrTTorqueSensorMeasRange^.T_Config.tDelayOff								:=ptrTTorqueSensorMeasRange^.T_Config.tDelayOff;
ptrTTorqueSensorMeasRange^.T_Config.tDelayOn								:=T#100ms;
ptrTTorqueSensorMeasRange^.T_CtrleCyl.T_Standard.tDelayAfterSensorOff			:=ptrTTorqueSensorMeasRange^.T_CtrleCyl.T_Standard.tDelayAfterSensorOff;
ptrTTorqueSensorMeasRange^.T_CtrleCyl.T_Standard.tDelayAfterSensorOn			:=ptrTTorqueSensorMeasRange^.T_CtrleCyl.T_Standard.tDelayAfterSensorOn;
ptrTTorqueSensorMeasRange^.T_CtrleCyl.T_Standard.tDelayActiv					:=ptrTTorqueSensorMeasRange^.T_CtrleCyl.T_Standard.tDelayActiv;
ptrTTorqueSensorMeasRange^.T_Config.tDelayPreOff								:=T#0s;
ptrTTorqueSensorMeasRange^.T_Config.tDelayPreOn								:=T#0s;

(* Config Sensor TorqueSensorControl *)
ptrTTorqueSensorControl^.iCylinderTpye											:=23;
ptrTTorqueSensorControl^.T_CtrleCyl.xFBActiv									:=T_Station_Work.TControl.xEnable;
ptrTTorqueSensorControl^.T_Config.xActivState									:=TRUE;
ptrTTorqueSensorControl^.T_Config.xCtrlePosOff									:=FALSE;
ptrTTorqueSensorControl^.T_Config.xCtrlePosOn									:=FALSE;
ptrTTorqueSensorControl^.T_Config.tTimeOut										:=T#0s;
ptrTTorqueSensorControl^.T_Config.tDelayOff										:=ptrTTorqueSensorControl^.T_Config.tDelayOff;
ptrTTorqueSensorControl^.T_Config.tDelayOn										:=T#100ms;
ptrTTorqueSensorControl^.T_CtrleCyl.T_Standard.tDelayAfterSensorOff				:=ptrTTorqueSensorControl^.T_CtrleCyl.T_Standard.tDelayAfterSensorOff;
ptrTTorqueSensorControl^.T_CtrleCyl.T_Standard.tDelayAfterSensorOn				:=ptrTTorqueSensorControl^.T_CtrleCyl.T_Standard.tDelayAfterSensorOn;
ptrTTorqueSensorControl^.T_CtrleCyl.T_Standard.tDelayActiv						:=ptrTTorqueSensorControl^.T_CtrleCyl.T_Standard.tDelayActiv;
ptrTTorqueSensorControl^.T_Config.tDelayPreOff									:=T#0s;
ptrTTorqueSensorControl^.T_Config.tDelayPreOn									:=T#0s;

(* Config Bubbler Axis *)
ptrTAxisBubbler^.T_Config_Gen.iTyp:=5; (* Bubbler Axis-->DC-Achse für Rührwerk *)
ptrTAxisBubbler^.T_Config_Gen.sDeviceFileName:='EC-MAX2611W_Bubbler_St1_KL2552';
(* Config Feedpump Axis *)
ptrTAxisFeedPump^.T_Config_Gen.iTyp:=6; (* Feedpump Axis-->DC-Achse für Förderpumpe *)
ptrTAxisFeedPump^.T_Config_Gen.sDeviceFileName:='EC-MAX2611W_Feedpump_St1_KL2552';
END_ACTION
ACTION HW_Axis_DC:
(******************************************************************************************************************************************)
(****************************				            Axis Bubbler Motion                                                *****************************)
(******************************************************************************************************************************************)
fbBubbler(	T_Axis_DC:= ptrTAxisBubbler^,
			usiStatusWord:= stBubblerDataIN.usiStatusWord,
			usiControlWord:= stBubblerDataOUT.usiControlWord,
			iDataOut:= stBubblerDataOUT.iDataOut,
			iDataIn:= stBubblerDataIN.iDataIn,
			T_HDD:= T_HDD);
(******************************************************************************************************************************************)
(****************************				            Axis Feedpump Motion                                          *****************************)
(******************************************************************************************************************************************)
fbFeedpump(	T_Axis_DC:= ptrTAxisFeedPump^,
			usiStatusWord:= stFeedpumpINData.usiStatusWord,
			usiControlWord:= stFeedpumpOUTData.usiControlWord,
			iDataOut:= stFeedpumpOUTData.iDataOut,
			iDataIn:= stFeedpumpINData.iDataIn,
			T_HDD:= T_HDD);
END_ACTION
ACTION HW_AxisS:
(******************************************************************************************************************************************)
(****************************			            Axis Tool Spindle Live Values                                     *****************************)
(******************************************************************************************************************************************)
CASE T_ExchgParam.bToolSpindleActive OF
1:	(* Maxon Spindel *)
	IF (T_Station_Parameter.T_TorqueSystem.rGearRatioGearBox <> 0.0) AND (T_Station_Parameter.T_TorqueSystem.rGearRatioSpindleMotor <> 0.0) THEN
		ptrTAxisS^.T_CtrleSingle.lrScaleFactor:=	1.0/ T_Station_Parameter.T_TorqueSystem.rGearRatioSpindleMotor / T_Station_Parameter.T_TorqueSystem.rGearRatioGearBox;
	ELSE
		ptrTAxisS^.T_CtrleSingle.lrScaleFactor:=1.8315;	(* Gilt für 60W Motoren *)
	END_IF;
	fbAxisToolSpindleSLiveValues(	uiActualTorque:= IuiActualTorqueAxisS,
								arxDigitalInput:= ,
								T_Axis:= ptrTAxisS^,
								T_AxisRefIn:= stSRefIn);
2:	(* Beckhoff Spindel L *)
	ptrTAxisS^.T_CtrleSingle.lrScaleFactor:=6.0;
	fbAxisToolSpindleSLiveValues(	uiActualTorque:= IuiActualTorqueAxisS,
								arxDigitalInput:= ,
								T_Axis:= ptrTAxisS^,
								T_AxisRefIn:= stS2RefIn);
3:	(* Beckhoff Spindel M *)
	ptrTAxisS^.T_CtrleSingle.lrScaleFactor:=6.0;
	fbAxisToolSpindleSLiveValues(	uiActualTorque:= IuiActualTorqueAxisS,
								arxDigitalInput:= ,
								T_Axis:= ptrTAxisS^,
								T_AxisRefIn:= stS3RefIn);
END_CASE;
(******************************************************************************************************************************************)
(****************************		                           Axis Tool Spindle Motion                                          *****************************)
(******************************************************************************************************************************************)
CASE T_ExchgParam.bToolSpindleActive OF
1:	(* Maxon Spindel *)
	fbAxisToolSpindleS(	xHWLimitPos:= FALSE,
						xHWLimitNeg:= FALSE,
						xRefHoming:= FALSE,
						wInputState:=IwInputState_S1_Axis,
						wPosLimitSwitchBit:=0,
						wNegLimitSwitchBit:=0,
						lrNullPointOffset:=0.0,
						IxSoftLimitMaxMonitoring:=,
						T_Axis:= ptrTAxisS^,
						T_AxisRefIn:= stSRefIn,
						T_AxisRefOut:= stSRefOut,
						T_HDD:= T_HDD);
2:	(* Beckhoff Spindel L *)
	fbAxisToolSpindleS(	xHWLimitPos:= FALSE,
						xHWLimitNeg:= FALSE,
						xRefHoming:= FALSE,
						wInputState:=IwInputState_S2_Axis,
						wPosLimitSwitchBit:=0,
						wNegLimitSwitchBit:=0,
						lrNullPointOffset:=0.0,
						IxSoftLimitMaxMonitoring:=,
						T_Axis:= ptrTAxisS^,
						T_AxisRefIn:= stS2RefIn,
						T_AxisRefOut:= stS2RefOut,
						T_HDD:= T_HDD);
3:	(* Beckhoff Spindel M *)
	fbAxisToolSpindleS(	xHWLimitPos:= FALSE,
						xHWLimitNeg:= FALSE,
						xRefHoming:= FALSE,
						wInputState:=IwInputState_S3_Axis,
						wPosLimitSwitchBit:=0,
						wNegLimitSwitchBit:=0,
						lrNullPointOffset:=0.0,
						IxSoftLimitMaxMonitoring:=,
						T_Axis:= ptrTAxisS^,
						T_AxisRefIn:= stS3RefIn,
						T_AxisRefOut:= stS3RefOut,
						T_HDD:= T_HDD);
END_CASE;
(******************************************************************************************************************************************)
(****************************		             Count Rotation Time of the Spindel                                     *****************************)
(******************************************************************************************************************************************)
CASE T_ExchgParam.bToolSpindleActive OF
1:	(* Maxon Spindel *)
	IF NOT(ptrTAxisS^.T_CtrleSingle.xNotMoving) AND NOT(ptrTAxisS^.T_CtrleSingle.xErr) THEN
		TONTickTime(IN:=TRUE,PT:=T#1s);
		IF TONTickTime.Q THEN
			TONTickTime(IN:=FALSE);
			T_Station_Work.THWWorkStation.TCtrlWork.tSpindelActiveRotationTime:=T_Station_Work.THWWorkStation.TCtrlWork.tSpindelActiveRotationTime + T#1s;
			IF T_Station_Work.THWWorkStation.TCtrlWork.tSpindelActiveRotationTime >= T#86400s THEN
				IF (T_Station_Work.THWWorkStation.TCtrlWork.iSpindelActiveRotationDay < 32767) THEN
					T_Station_Work.THWWorkStation.TCtrlWork.iSpindelActiveRotationDay:=T_Station_Work.THWWorkStation.TCtrlWork.iSpindelActiveRotationDay + 1;
				END_IF;
				T_Station_Work.THWWorkStation.TCtrlWork.tSpindelActiveRotationTime:=T#0s;
			END_IF;
		END_IF;
	ELSE
		TONTickTime(IN:=FALSE);
	END_IF;
2:	(* Beckhoff Spindel L *)
	IF NOT(ptrTAxisS^.T_CtrleSingle.xNotMoving) AND NOT(ptrTAxisS^.T_CtrleSingle.xErr) THEN
		TONTickTime(IN:=TRUE,PT:=T#1s);
		IF TONTickTime.Q THEN
			TONTickTime(IN:=FALSE);
			T_Station_Work.THWWorkStation.TCtrlWork.tSpindel2ActiveRotationTime:=T_Station_Work.THWWorkStation.TCtrlWork.tSpindel2ActiveRotationTime + T#1s;
			IF T_Station_Work.THWWorkStation.TCtrlWork.tSpindel2ActiveRotationTime >= T#86400s THEN
				IF (T_Station_Work.THWWorkStation.TCtrlWork.iSpindel2ActiveRotationDay < 32767) THEN
					T_Station_Work.THWWorkStation.TCtrlWork.iSpindel2ActiveRotationDay:=T_Station_Work.THWWorkStation.TCtrlWork.iSpindel2ActiveRotationDay + 1;
				END_IF;
				T_Station_Work.THWWorkStation.TCtrlWork.tSpindel2ActiveRotationTime:=T#0s;
			END_IF;
		END_IF;
	ELSE
		TONTickTime(IN:=FALSE);
	END_IF;
3:	(* Beckhoff Spindel M *)
	IF NOT(ptrTAxisS^.T_CtrleSingle.xNotMoving) AND NOT(ptrTAxisS^.T_CtrleSingle.xErr) THEN
		TONTickTime(IN:=TRUE,PT:=T#1s);
		IF TONTickTime.Q THEN
			TONTickTime(IN:=FALSE);
			T_Station_Work.THWWorkStation.TCtrlWork.tSpindel3ActiveRotationTime:=T_Station_Work.THWWorkStation.TCtrlWork.tSpindel3ActiveRotationTime + T#1s;
			IF T_Station_Work.THWWorkStation.TCtrlWork.tSpindel3ActiveRotationTime >= T#86400s THEN
				IF (T_Station_Work.THWWorkStation.TCtrlWork.iSpindel3ActiveRotationDay < 32767) THEN
					T_Station_Work.THWWorkStation.TCtrlWork.iSpindel3ActiveRotationDay:=T_Station_Work.THWWorkStation.TCtrlWork.iSpindel3ActiveRotationDay + 1;
				END_IF;
				T_Station_Work.THWWorkStation.TCtrlWork.tSpindel3ActiveRotationTime:=T#0s;
			END_IF;
		END_IF;
	ELSE
		TONTickTime(IN:=FALSE);
	END_IF;
END_CASE;
END_ACTION
ACTION HW_AxisZ:
(******************************************************************************************************************************************)
(*******************************				         Axis Z Live Values                                              *********************************)
(******************************************************************************************************************************************)
fbAxisZLiveValues(	uiActualTorque:= IuiActualTorqueAxisZ,
					arxDigitalInput:= ,
					T_Axis:= ptrTAxisZ^,
					T_AxisRefIn:= stZRefIn);
(******************************************************************************************************************************************)
(*********************************				            Axis Z Motion                                            ********************************)
(******************************************************************************************************************************************)

(*******************************            START: Manuelle Schleppabstandsüberwachung, da mit dem neuen Regler keine Überwachung mehr in der NC Ebene steht        ************************************************)
lrCtrlSpeed:=ABS(DINT_TO_LREAL(T_Z_St1_Ctrle.diVelocityCommandValue)/558349.25);	(* Soll Geschwindigkeit *)
lrActualSpeed:=ABS(ptrTAxisZ^.T_LiveValue.lrActualVelocity);								(* Ist Geschwindigkeit *)
lrCheckSpeed:=0.0;
IF (lrCtrlSpeed <= 1.0) AND (lrCtrlSpeed <> 0.0) THEN
	lrCheckSpeed:=0.5;
ELSIF (lrCtrlSpeed <= 10.0) AND (lrCtrlSpeed <> 0.0) THEN
	lrCheckSpeed:=2.0;
ELSIF (lrCtrlSpeed <= 100.0) AND (lrCtrlSpeed <> 0.0) THEN
	lrCheckSpeed:=10.0;
ELSIF (lrCtrlSpeed > 100.0) AND (lrCtrlSpeed <> 0.0) THEN
	lrCheckSpeed:=20.0;
END_IF;
lrCalcSpeed:=lrCtrlSpeed - lrActualSpeed;
IF (lrCheckSpeed <> 0.0) THEN
	IF (lrCalcSpeed >= lrCheckSpeed) THEN
		xZMovementNOK:=TRUE;
	ELSE
		xZMovementNOK:=FALSE;
	END_IF;
ELSE
	xZMovementNOK:=FALSE;
END_IF;
TONCheckMovement(IN:=xZMovementNOK,PT:=T#0.5s);
IF TONCheckMovement.Q THEN	(* Überwachen falls um diese Zeit die Geschwindigkeitsänderung zwischen Soll und Ist ansteht, dann muss der Schleppabstandsfehler erscheinen *)
	diCounterTest:=diCounterTest + 1;
	IF NOT(ptrTAxisZ^.T_CtrleSingle.xExecute) AND (ptrTAxisZ^.T_CtrleSingle.iFunction <> 5) THEN
		ptrTAxisZ^.T_CtrleSingle.iFunction:=5;
		ptrTAxisZ^.T_CtrleSingle.xExecute:=TRUE;
		gxZFollowDistanceError:=TRUE;
	END_IF;
END_IF;
(*******************************            ENDE: Manuelle Schleppabstandsüberwachung, da mit dem neuen Regler keine Überwachung mehr in der NC Ebene steht        ************************************************)

fbAxisZ(		xHWLimitPos:= FALSE,
			xHWLimitNeg:= FALSE,
			xRefHoming:= T_Station_Parameter.T_AxisState.xReferencedZAxis, (* Absolut Encoder, daher kein Ref.Sensor *)
			wInputState:=IwInputState_Z_Axis,
			wPosLimitSwitchBit:=ptrTAxisZ^.T_Config_Gen.wPosLimitSwitchBit,
			wNegLimitSwitchBit:=ptrTAxisZ^.T_Config_Gen.wNegLimitSwitchBit,
			lrNullPointOffset:=0.0,
			IxSoftLimitMaxMonitoring:=FALSE,
			T_Axis:= ptrTAxisZ^,
			T_AxisRefIn:= stZRefIn,
			T_AxisRefOut:= stZRefOut,
			T_HDD:= T_HDD);
END_ACTION
ACTION HW_CylBrakeReleaseZAxis:
(******************************************************************************************************************************************)
(********************************   		      Ventil für Bremse lösen der Z Achse                  ********************************)
(******************************************************************************************************************************************)
fbCylTBrakeReleaseZAxis(	xCtrlePosOn:= IxBrakeReleaseZAxis,
							xCtrlePosOff:=  FALSE,
							T_Cylinder:= ptrTCylBrakeReleaseZAxis^);
QxCylBrakeReleaseZAxis_Open:=fbCylTBrakeReleaseZAxis.xCylinderOn;	(* Ventil QxCylBrakeReleaseZ1Axis_Open-->Ventil für Bremszylinder der Z Achse für Bremse lösen *)
QxCylBrakeReleaseZAxis_Close:=fbCylTBrakeReleaseZAxis.xCylinderOff;	(* Ventil QxCylBrakeReleaseZ1Axis_Close-->Ventil für Bremszylinder der Z Achse für Bremse Aktivieren *)
END_ACTION
ACTION HW_CylToolDeflection:
(******************************************************************************************************************************************)
(****************************				          Cylinder Tool Deflection                                       *****************************)
(******************************************************************************************************************************************)
CASE T_ExchgParam.bToolSpindleActive OF
	1:	(* Maxon Spindel *)
	FBCalcSpindleForce(	rForcePistonIn:= ptrTCylToolDeflection^.T_CtrleCyl.T_Analog.rForceIn + T_Station_Parameter.T_Fct_SpindleCalibration.arOffsetToolDeflection[1],
						rPistonDiameterD1:= T_Station_Parameter.T_SpindleSystem.rPistonDiameterD1,
						rPistonDiameterD2:= T_Station_Parameter.T_SpindleSystem.rPistonDiameterD2,
						rMaxAirpressure:= T_Station_Parameter.T_SpindleSystem.rMaxServoAirPressure,
						rMaxServoVoltage:=T_Station_Parameter.T_SpindleSystem.rMaxServoVoltage);
	T_Station_Parameter.T_SpindleSystem.rMaxDeflectionForce:=FBCalcSpindleForce.rSetMaxForce - T_Station_Parameter.T_Fct_SpindleCalibration.arOffsetToolDeflection[1];
	ptrTCylToolDeflection^.T_CtrleCyl.T_Analog.iAnalogIN:=FBCalcSpindleForce.iAnalogOutput;
	ptrTCylToolDeflection^.T_CtrleCyl.T_Analog.rForceOut:=FBCalcSpindleForce.rForcePistonOut;
	fbCylToolDeflection(	xCtrlePosOn:=IxToolDeflection,
						xCtrlePosOff:= FALSE,
						iAnalogIn:= ptrTCylToolDeflection^.T_CtrleCyl.T_Analog.iAnalogIN,
						T_Cylinder:= ptrTCylToolDeflection^);
	QiAToolDeflection_SM:=fbCylToolDeflection.iAnalogOut;	(* Servoventil QiAToolDeflection_SM_St1 (2Bar) *)
	ptrTCylToolDeflection^.T_CtrleCyl.T_Analog.iAnalogOut:=fbCylToolDeflection.iAnalogOut;
2:	(* Beckhoff Spindel L *)
	FBCalcSpindleForce(	rForcePistonIn:= ptrTCylToolDeflection^.T_CtrleCyl.T_Analog.rForceIn + T_Station_Parameter.T_Fct_SpindleCalibration.arOffsetToolDeflection[1],
						rPistonDiameterD1:= T_Station_Parameter.T_SpindleSystem_L.rPistonDiameterD1,
						rPistonDiameterD2:= T_Station_Parameter.T_SpindleSystem_L.rPistonDiameterD2,
						rMaxAirpressure:= T_Station_Parameter.T_SpindleSystem_L.rMaxServoAirPressure,
						rMaxServoVoltage:=T_Station_Parameter.T_SpindleSystem_L.rMaxServoVoltage);
	T_Station_Parameter.T_SpindleSystem_L.rMaxDeflectionForce:=FBCalcSpindleForce.rSetMaxForce - T_Station_Parameter.T_Fct_SpindleCalibration.arOffsetToolDeflection[1];
	ptrTCylToolDeflection^.T_CtrleCyl.T_Analog.iAnalogIN:=FBCalcSpindleForce.iAnalogOutput;
	ptrTCylToolDeflection^.T_CtrleCyl.T_Analog.rForceOut:=FBCalcSpindleForce.rForcePistonOut;
	fbCylToolDeflection(	xCtrlePosOn:=IxToolDeflection,
						xCtrlePosOff:= FALSE,
						iAnalogIn:= ptrTCylToolDeflection^.T_CtrleCyl.T_Analog.iAnalogIN,
						T_Cylinder:= ptrTCylToolDeflection^);
	QiAToolTorqueOverload_SM:=fbCylToolDeflection.iAnalogOut;	(* Servoventil QiAToolTorqueOverload_SM_St1 (8Bar) *)
	ptrTCylToolDeflection^.T_CtrleCyl.T_Analog.iAnalogOut:=fbCylToolDeflection.iAnalogOut;
	QiAToolDeflection_SM:=0;
3:	(* Beckhoff Spindel M *)
	FBCalcSpindleForce(	rForcePistonIn:= ptrTCylToolDeflection^.T_CtrleCyl.T_Analog.rForceIn + T_Station_Parameter.T_Fct_SpindleCalibration.arOffsetToolDeflection[1],
						rPistonDiameterD1:= T_Station_Parameter.T_SpindleSystem_M.rPistonDiameterD1,
						rPistonDiameterD2:= T_Station_Parameter.T_SpindleSystem_M.rPistonDiameterD2,
						rMaxAirpressure:= T_Station_Parameter.T_SpindleSystem_M.rMaxServoAirPressure,
						rMaxServoVoltage:=T_Station_Parameter.T_SpindleSystem_M.rMaxServoVoltage);
	T_Station_Parameter.T_SpindleSystem_M.rMaxDeflectionForce:=FBCalcSpindleForce.rSetMaxForce - T_Station_Parameter.T_Fct_SpindleCalibration.arOffsetToolDeflection[1];
	ptrTCylToolDeflection^.T_CtrleCyl.T_Analog.iAnalogIN:=FBCalcSpindleForce.iAnalogOutput;
	ptrTCylToolDeflection^.T_CtrleCyl.T_Analog.rForceOut:=FBCalcSpindleForce.rForcePistonOut;
	fbCylToolDeflection(	xCtrlePosOn:=IxToolDeflection,
						xCtrlePosOff:= FALSE,
						iAnalogIn:= ptrTCylToolDeflection^.T_CtrleCyl.T_Analog.iAnalogIN,
						T_Cylinder:= ptrTCylToolDeflection^);
	QiAToolDeflection_SM:=fbCylToolDeflection.iAnalogOut;	(* Servoventil QiAToolDeflection_SM_St1 (2Bar) *)
	ptrTCylToolDeflection^.T_CtrleCyl.T_Analog.iAnalogOut:=fbCylToolDeflection.iAnalogOut;
	QiAToolTorqueOverload_SM:=0;
END_CASE;
END_ACTION
ACTION HW_CylWorkpieceClamp:
(******************************************************************************************************************************************)
(********************************   		       Ventil für Werkstückfxierungszylinder                  ********************************)
(******************************************************************************************************************************************)
fbCylWorkpieceClamp(	xCtrlePosOn:= 	IxUpperToolGuide_WorkpieceClamped, 	(* Sensor für Überwachung der Werkstückfixierung *)
						xCtrlePosOff:=  FALSE,
						T_Cylinder:= ptrTCylWorkpieceClamp^);
QxCylWorkpieceClamp_Close:=fbCylWorkpieceClamp.xCylinderOn;	(* Ventil QxCylWorkpieceClamp_Close-->Ventil für Werkstückfixierzylinder schliessen *)
QxCylWorkpieceClamp_Open:=fbCylWorkpieceClamp.xCylinderOff;	(* Ventil QxCylWorkpieceClamp_Open-->Ventil für Werkstückfixierzylinder öffnen *)
END_ACTION
ACTION HW_ToolTorqueHC:
(******************************************************************************************************************************************)
(****************************				          Cylinder Torque HC                                                  *****************************)
(******************************************************************************************************************************************)
CASE T_ExchgParam.bToolSpindleActive OF
1:	(* Maxon Spindel *)
	FBTorqueLevelAirPressureAnalog_HC(	xActiveWorkProcess:= T_Station_Work.THWWorkStation.TCtrlWork.xActiveProcess_CylToolTorqueHC,
										xBlockOutput:= T_Station_Work.THWWorkStation.TCtrlWork.xBlockOutput_CylToolTorqueHC,
										rForceIn:= ptrTCylToolTorqueHC^.T_CtrleCyl.T_Analog.rForceIn + T_Station_Parameter.T_Fct_SpindleCalibration.arOffsetToolTorque[1],
										T_Station_Parameter:= T_Station_Parameter,
										lrZ1ActualPosition:= ptrTAxisZ^.T_LiveValue.lrActualPosition,
										xCylHCActive:=TRUE,
										TCylTorque:= ptrTCylToolTorqueHC^,
										iAnalogOutput=> ptrTCylToolTorqueHC^.T_CtrleCyl.T_Analog.iAnalogIN,
										rForceOut=> ptrTCylToolTorqueHC^.T_CtrleCyl.T_Analog.rForceOut);
	T_Station_Parameter.T_TorqueSystem.rMaxTorque_HC:=FBTorqueLevelAirPressureAnalog_HC.rMaxTorque - T_Station_Parameter.T_Fct_SpindleCalibration.arOffsetToolTorque[1];

	fbCylToolTorqueHC(	xCtrlePosOn:=ptrTCylToolTorqueHC^.T_CtrleCyl.xStatePosOn,
						xCtrlePosOff:= FALSE,
						iAnalogIn:= ptrTCylToolTorqueHC^.T_CtrleCyl.T_Analog.iAnalogIN,
						T_Cylinder:= ptrTCylToolTorqueHC^);
	QiAToolTorqueHC_SM:=fbCylToolTorqueHC.iAnalogOut;
	ptrTCylToolTorqueHC^.T_CtrleCyl.T_Analog.iAnalogOut:=fbCylToolTorqueHC.iAnalogOut;
2,3:	(* Beckhoff Spindel *)
	QiAToolTorqueHC_SM:=0;
	ptrTCylToolTorqueHC^.T_CtrleCyl.T_Analog.iAnalogOut:=0;
END_CASE;
END_ACTION
ACTION HW_ToolTorqueOverload:
(******************************************************************************************************************************************)
(****************************				    Cylinder Torque Overload                                           *****************************)
(******************************************************************************************************************************************)
CASE T_ExchgParam.bToolSpindleActive OF
1:	(* Maxon Spindel *)
	rCalcForceIn:=ptrTCylToolTorqueOverload^.T_CtrleCyl.T_Analog.rForceIn - ptrTCylToolTorqueHC^.T_CtrleCyl.T_Analog.rForceIn + T_Station_Parameter.T_Fct_SpindleCalibration.arOffsetToolTorque[1];
	IF (rCalcForceIn < 0.0) THEN
		rCalcForceIn:=0.0;
	END_IF;
	FBTorqueLevelAirPressureAnalog_Overload(	xActiveWorkProcess:= FALSE,
											xBlockOutput:= FALSE,
											rForceIn:= rCalcForceIn,
											T_Station_Parameter:= T_Station_Parameter,
											lrZ1ActualPosition:= ptrTAxisZ^.T_LiveValue.lrActualPosition,
											xCylHCActive:=FALSE,
											TCylTorque:= ptrTCylToolTorqueOverload^,
											iAnalogOutput=> ptrTCylToolTorqueOverload^.T_CtrleCyl.T_Analog.iAnalogIN,
											rForceOut=> ptrTCylToolTorqueOverload^.T_CtrleCyl.T_Analog.rForceOut);
	T_Station_Parameter.T_TorqueSystem.rMaxTorque_HCOver:=FBTorqueLevelAirPressureAnalog_Overload.rMaxTorque - T_Station_Parameter.T_Fct_SpindleCalibration.arOffsetToolTorque[1] +
														     ((T_Station_Parameter.T_OnlineChange.rTorqueLevelHC + T_Station_Parameter.T_OnlineChange.rTorqueLevelHC) /2.0);
	fbCylToolTorqueOverload(	xCtrlePosOn:=ptrTCylToolTorqueOverload^.T_CtrleCyl.xStatePosOn,
							xCtrlePosOff:= FALSE,
							iAnalogIn:= ptrTCylToolTorqueOverload^.T_CtrleCyl.T_Analog.iAnalogIN,
							T_Cylinder:= ptrTCylToolTorqueOverload^);
	QiAToolTorqueOverload_SM:=fbCylToolTorqueOverload.iAnalogOut;
	ptrTCylToolTorqueOverload^.T_CtrleCyl.T_Analog.iAnalogOut:=fbCylToolTorqueOverload.iAnalogOut;
2,3:	(* Beckhoff Spindel *)
	QiAToolTorqueOverload_SM:=0;
	ptrTCylToolTorqueOverload^.T_CtrleCyl.T_Analog.iAnalogOut:=0;
END_CASE;
END_ACTION
ACTION HW_TorqueOverloadSensor:
(******************************************************************************************************************************************)
(****************************  		       Sensor für Drehmomentüberlastdetektion                  ********************************)
(******************************************************************************************************************************************)
IF NOT(xInitState) THEN
	xInitState:=TRUE;
	udiTorqueOverloadCounterValue:=gudiTorqueOverloadCounterValueSt1;
END_IF;
TOFSetOutput(IN:=(udiTorqueOverloadCounterValue<>gudiTorqueOverloadCounterValueSt1),PT:=T#2s);
IF (udiTorqueOverloadCounterValue<>gudiTorqueOverloadCounterValueSt1) THEN
	xInitState:=FALSE;
END_IF;
ptrTSensorTorqueOverload^.T_CtrleCyl.xStatePosOn:=IxTorqueOverload OR TOFSetOutput.Q;
ptrTSensorTorqueOverload^.T_CtrleCyl.xDone:=TRUE;
END_ACTION
ACTION HW_TorqueSensor:
(******************************************************************************************************************************************)
(****************************  		       Analog Sensor für Drehmomentdetektion                  ********************************)
(******************************************************************************************************************************************)
CASE T_ExchgParam.bToolSpindleActive OF
1:	(* Maxon Spindel *)
	IF (T_Station_Parameter.T_TorqueSystem.rTorqueScaleFactor <> 0.0) THEN
		T_Station_Work.THWWorkStation.TSensorTorque.T_CtrleCyl.T_Analog.rPosIn:=	(INT_TO_REAL(IiAToolTorque) /
																				T_Station_Parameter.T_TorqueSystem.rTorqueScaleFactor)
																				* T_Station_Parameter.T_TorqueSystem.rMeasureDistance;
	ELSE
		T_Station_Work.THWWorkStation.TSensorTorque.T_CtrleCyl.T_Analog.rPosIn:=	INT_TO_REAL(IiAToolTorque);
	END_IF;

	ptrTCylToolTorqueHC^.T_CtrleCyl.xStatePosOn:=	T_Station_Work.THWWorkStation.TSensorTorque.T_CtrleCyl.T_Analog.rPosIn >
												T_Station_Parameter.T_TorqueSystem.rTorquePosition_HC;

	ptrTCylToolTorqueOverload^.T_CtrleCyl.xStatePosOn:=	T_Station_Work.THWWorkStation.TSensorTorque.T_CtrleCyl.T_Analog.rPosIn >
													T_Station_Parameter.T_TorqueSystem.rTorquePosition_HCOverload;
END_CASE;

IF (ii <= 0) THEN
	ii:=1;
END_IF;
IF TStation_Work_St1.THWWorkStation.TAxisS.T_CtrleSingle.xExecute AND TStation_Work_St1.THWWorkStation.TCylToolTorqueHC.T_CtrleCyl.T_Analog.xActiv THEN
	rDefaultValue:=TStation_Work_St1.THWWorkStation.TSensorTorque.T_CtrleCyl.T_Analog.rPosIn * 25.4;
END_IF;
garRockerMeasureValue[ii]:=TStation_Work_St1.THWWorkStation.TSensorTorque.T_CtrleCyl.T_Analog.rPosIn * 25.4;
ii:=ii+1;
IF (ii > 200) THEN
	grRockerMinValue:=garRockerMeasureValue[1];
	grRockerMaxValue:=garRockerMeasureValue[1];
	rQualitySum:=0;
	FOR jj:=1 TO 200 DO
		IF (garRockerMeasureValue[jj] < grRockerMinValue) THEN
			grRockerMinValue:=garRockerMeasureValue[jj];
		END_IF;
		IF (garRockerMeasureValue[jj] > grRockerMaxValue) THEN
			grRockerMaxValue:=garRockerMeasureValue[jj];
		END_IF;
		rQualitySum:=rQualitySum + garRockerMeasureValue[jj];
	END_FOR;
	rQualityArea:=200.0 * grRockerMaxValue;
	IF (rQualityArea <> 0.0) THEN
		rQuality:=100.0/rQualityArea*rQualitySum;
	ELSE
		rQuality:=100.0;
	END_IF;
	IF (rQuality < 0.0) THEN
		rQuality:=0.0;
	ELSIF (rQuality > 100.0) THEN
		rQuality:=100.0;
	END_IF;
	ii:=1;
END_IF;
grRockerQuality:=rQuality;
grRockerAmplitude:=(100.0 / ((T_NovRam.T_Parameter.T_StationWork[gciStationSt1].T_TorqueSystem.rTorquePosition_HC * 25.4) - rDefaultValue)) * (grRockerMaxValue - rDefaultValue);
IF (grRockerAmplitude < 0.0) THEN
	grRockerAmplitude:=0.0;
ELSIF (grRockerAmplitude > 100.0) THEN
	grRockerAmplitude:=100.0;
END_IF;
IF NOT(TStation_Work_St1.THWWorkStation.TAxisS.T_CtrleSingle.xNotMoving) THEN
	TONWaitCycle(IN:=TRUE,PT:=T#2s);
	IF NOT(xFirstTime) AND TONWaitCycle.Q THEN
		xFirstTime:=TRUE;
		grRockerAmplitudeMin:=grRockerAmplitude;
		grRockerAmplitudeMax:=grRockerAmplitude;
		grRockerQualityMin:=grRockerQuality;
		grRockerQualityMax:=grRockerQuality;
	END_IF;
	IF TONWaitCycle.Q THEN
		IF (grRockerAmplitude < grRockerAmplitudeMin) THEN
			grRockerAmplitudeMin:=grRockerAmplitude;
		END_IF;
		IF (grRockerAmplitude > grRockerAmplitudeMax) THEN
			grRockerAmplitudeMax:=grRockerAmplitude;
		END_IF;
		IF (grRockerQuality < grRockerQualityMin) THEN
			grRockerQualityMin:=grRockerQuality;
		END_IF;
		IF (grRockerQuality > grRockerQualityMax) THEN
			grRockerQualityMax:=grRockerQuality;
		END_IF;
	ELSE
		grRockerAmplitudeMin:=0;
		grRockerAmplitudeMax:=0;
		grRockerQualityMin:=0;
		grRockerQualityMax:=0;
		gdiRockerCountHC:=0;
		gdiRockerCountHCTime:=0;
	END_IF;
ELSE
	TONWaitCycle(IN:=FALSE);
	xFirstTime:=FALSE;
END_IF;
TONCalcImpuls(IN:=ptrTCylToolTorqueHC^.T_CtrleCyl.xStatePosOn,PT:=T#99999s);
IF ptrTCylToolTorqueHC^.T_CtrleCyl.xStatePosOn THEN
	IF NOT(xInitCountHC) THEN
		xInitCountHC:=TRUE;
		gdiRockerCountHC:=gdiRockerCountHC+1;
	END_IF;
	gdiRockerCountHCTime:=TIME_TO_DINT(TONCalcImpuls.ET);
	xTorqueActive:=TRUE;
ELSE
	xInitCountHC:=FALSE;
	IF xTorqueActive THEN
		xTorqueActive:=FALSE;
		IF (gdiRockerCountHCTime = 0) THEN
			gdiRockerCountHCTime:=2;
		END_IF;
	END_IF;
END_IF;
grRockerPosition:=(100.0 / ((T_NovRam.T_Parameter.T_StationWork[gciStationSt1].T_TorqueSystem.rTorquePosition_HC * 25.4) - rDefaultValue)) *
				((TStation_Work_St1.THWWorkStation.TSensorTorque.T_CtrleCyl.T_Analog.rPosIn * 25.4) - rDefaultValue);
IF (grRockerPosition < 0.0) THEN
	grRockerPosition:=0.0;
ELSIF (grRockerPosition > 100.0) THEN
	grRockerPosition:=100.0;
END_IF;
T_ExchgParam.T_StationCommon.rRockerAmplitude:=grRockerAmplitude;
T_ExchgParam.T_StationCommon.rRockerAmplitudeMin:=grRockerAmplitudeMin;
T_ExchgParam.T_StationCommon.rRockerAmplitudeMax:=grRockerAmplitudeMax;
T_ExchgParam.T_StationCommon.rRockerQuality:=grRockerQuality;
T_ExchgParam.T_StationCommon.rRockerQualityMin:=grRockerQualityMin;
T_ExchgParam.T_StationCommon.rRockerQualityMax:=grRockerQualityMax;
T_ExchgParam.T_StationCommon.rRockerPosition:=grRockerPosition;
T_ExchgParam.T_StationCommon.diRockerCountHC:=gdiRockerCountHC;
T_ExchgParam.T_StationCommon.diRockerCountHCTime:=gdiRockerCountHCTime;
END_ACTION
ACTION HW_TorqueSensor2:
(******************************************************************************************************************************************)
(****************************  		       Analog Sensor für Drehmomentdetektion                  ********************************)
(******************************************************************************************************************************************)
ptrTSensorTorque^.T_CtrleCyl.T_Analog.rPosIn:= ((INT_TO_REAL(IiAToolTorque2)/32767.0)*2000.0) - T_Station_Parameter.T_Fct_SpindleCalibration.arOffsetToolTorque[1];	(* Messbereich 0 - 2Nm-->2000mNm *)
IF (ptrTSensorTorque^.T_CtrleCyl.T_Analog.rPosIn <= 0.0) THEN
	ptrTSensorTorque^.T_CtrleCyl.T_Analog.rPosIn:=0.0;
END_IF;
ptrTSensorTorque^.T_CtrleCyl.xDone:=TRUE;

(* Drehmoment für Bearbeitung *)
ptrTSensorTorque^.T_CtrleCyl.xStatePosOn:=		ptrTSensorTorque^.T_CtrleCyl.T_Analog.rPosIn >=
												T_Station_Parameter.T_OnlineChange.rTorqueLevelHC;

(* Drehmoment für Ausfunken *)
ptrTSensorTorque^.T_CtrleCyl.xStatePosOn1:= 	ptrTSensorTorque^.T_CtrleCyl.T_Analog.rPosIn >=
												((T_Station_Parameter.T_OnlineChange.rTorqueLevelHC/100.0)*T_Station_Parameter.T_StProcess.rSparkOutTorqueLevel);

(* Drehmoment für Regler *)
ptrTSensorTorque^.T_CtrleCyl.xStatePosOff:=		(ptrTSensorTorque^.T_CtrleCyl.T_Analog.rPosIn >= 0.5);

CASE T_ExchgParam.bToolSpindleActive OF
2:	T_Station_Parameter.T_TorqueSystem_L.rActual_Torque:=	ptrTSensorTorque^.T_CtrleCyl.T_Analog.rPosIn;
3:	T_Station_Parameter.T_TorqueSystem_M.rActual_Torque:=	ptrTSensorTorque^.T_CtrleCyl.T_Analog.rPosIn;
END_CASE;
END_ACTION
ACTION HW_TorqueSensorControl:
(******************************************************************************************************************************************)
(****************************  		   Drehmomentsensor Überprüfung Funktionalität             ********************************)
(******************************************************************************************************************************************)
fbTorqueSensorControl(	xCtrlePosOn:= FALSE,
						xCtrlePosOff:= FALSE,
						T_Cylinder:= ptrTTorqueSensorControl^);
QxControlTorqueSensor:=fbTorqueSensorControl.xCylinder;
END_ACTION
ACTION HW_TorqueSensorMeasureRange:
(******************************************************************************************************************************************)
(****************************  		     Drehmomentsensor Messbreicheinstellung                  ********************************)
(******************************************************************************************************************************************)
fbTorqueSensorMeasRange(	xCtrlePosOn:= FALSE,
							xCtrlePosOff:= FALSE,
							T_Cylinder:= ptrTTorqueSensorMeasRange^);
QxMeasRangeTorqueSensor:=fbTorqueSensorMeasRange.xCylinder;
END_ACTION
ACTION HW_TSensorToolSpindle_L_Connect:
(******************************************************************************************************************************************)
(************************  		       Digitaler Sensor für Spindelkopf L angeschlossen                         ***************************)
(******************************************************************************************************************************************)
T_Station_Work.THWWorkStation.TSensorToolSpindle_L_Connect.T_CtrleCyl.xStatePosOff:=(IbTooSpindleActive = 1);
T_Station_Work.THWWorkStation.TSensorToolSpindle_L_Connect.T_CtrleCyl.xStatePosOn:=(IbTooSpindleActive = 2);
T_Station_Work.THWWorkStation.TSensorToolSpindle_L_Connect.T_CtrleCyl.xStatePosOn1:=(IbTooSpindleActive = 3);
END_ACTION
ACTION HW_ValveAirTable:
(******************************************************************************************************************************************)
(********************************   		               Ventil für Luft des Tisches                           ********************************)
(******************************************************************************************************************************************)
fbValveAirTable(		xCtrlePosOn:= FALSE,
					xCtrlePosOff:= FALSE,
					T_Cylinder:= ptrTValveAirTable^);
QxAirTable:=fbValveAirTable.xCylinder;	(* Ventil QxAirTable-->Ventil für die Luft des Tisches *)
END_ACTION
ACTION HW_ValveCleanNozzle:
(******************************************************************************************************************************************)
(******************************** 					 Ventil fuer die Reinigungsduese 			 ********************************)
(******************************************************************************************************************************************)
fbValveCleanNozzle(	xCtrlePosOn:= FALSE,
					xCtrlePosOff:= FALSE,
					T_Cylinder:= ptrTValveCleanNozzle^);
QxValveCleanNozzle:=fbValveCleanNozzle.xCylinder;	(* Ventil QxValveCleanNozzle-->Ventil fuer die Reinigungsduese *)
END_ACTION
ACTION HW_ValveVacuumTable:
(******************************************************************************************************************************************)
(********************************   		        Ventil fuer das Vakuum des Tisches                    ********************************)
(******************************************************************************************************************************************)
fbValveVacuumTable(		xCtrlePosOn:= FALSE,
							xCtrlePosOff:= FALSE,
							T_Cylinder:= ptrTValveVacuumTable^);
QxVacuumTable:=fbValveVacuumTable.xCylinder;	(* Ventil QxVacuumTable-->Ventil fuer das Vakuum des Tisches *)
END_ACTION

(* POU FB_HARDWARE/FBHW_AXIS_SINGLE, ST *)
FUNCTION_BLOCK FBHW_AXIS_SINGLE
VAR_INPUT
	xHWLimitPos:BOOL:=FALSE;
	xHWLimitNeg:BOOL:=FALSE;
	xRefHoming:BOOL:=FALSE;
	wInputState:WORD;
	lrNullPointOffset:LREAL;
	IxSoftLimitMaxMonitoring:BOOL;
	wPosLimitSwitchBit:WORD;
	wNegLimitSwitchBit:WORD;
	uiStateAxisZ2_KL2541:UINT;
END_VAR
VAR_OUTPUT
END_VAR
VAR_IN_OUT
	T_Axis:ST_AXIS;
	T_AxisRefIn:NCTOPLC_AXLESTRUCT;
	T_AxisRefOut:PLCTONC_AXLESTRUCT;
	T_HDD:ST_HDD;
END_VAR
VAR
(* Axis function block *)
	fbAxisReset:MC_Reset;
	fbAxisPower:MC_Power;
	fbAxisStop:MC_Stop;
	fbAxisMoveVelocity:MC_MoveVelocity;
	fbAxisMoveAbsolute:MC_MoveAbsolute;
	fbAxisMoveRelative:MC_MoveRelative;
	fbAxisMoveModulo:MC_MoveModulo;
	fbAxisHoming:MC_Home;
	fbAxisSetOverride:MC_SetOverride;
	fbAxisSetPosition:MC_SetActualPosition;
	fbAxisNewPosAndVel:MC_NewPosAndVelo;
	fbAxisSetReferenceFlag:MC_SetReferenceFlag;
	fbDefaultAxisPara:FBDefaultAxisValue;
	fbAdsWrite:ADSWRITE;
	fbADS_ReadWriteString:ADSRDWRTEX;
	fbExtSetPointGenDisable:MC_ExtSetPointGenDisable;
	fbExtSetPointGenEnable:MC_ExtSetPointGenEnable;
(* variable *)
	xConfirmResetFB:BOOL:=FALSE;
	xResetAxis:BOOL:=FALSE;
	xPowerOn:BOOL:=FALSE;
	xPowerOff:BOOL:=FALSE;
	xStop:BOOL:=FALSE;
	xMoveVel:BOOL:=FALSE;
	iDirectionVel:INT:=1;
	rVelocity:REAL:=0;
	xMoveAbs:BOOL:=FALSE;
	xMoveRel:BOOL:=FALSE;
	xMoveModulo:BOOL:=FALSE;
	xHoming:BOOL:=FALSE;
	xOverride:BOOL:=FALSE;
	xSetPosition:BOOL:=FALSE;
	xNewVelocity:BOOL:=FALSE;
	xNewPosition:BOOL:=FALSE;
	xCalcAngleRefIndex: BOOL:=FALSE;
	xSetReferenceFlag:BOOL:=FALSE;
	xResetReferenceFlag:BOOL:=FALSE;
	xDefaultAxisParameter:BOOL:=FALSE;
	xSendAxisParameter:BOOL:=FALSE;
	iPtrAxisParameter:INT:=0;
	xSendAxisString:BOOL:=FALSE;
	sSendAxis:STRING:='';
	sReturnAxis:STRING:='';
	iStepSendPara:INT:=0;
	xRestoreAxisPower:BOOL:=FALSE;
	iStepFile:INT:=0;
	xCtrlePositionOn:BOOL:=FALSE;
	xCtrlePositionOff:BOOL:=FALSE;
	xOscillation:BOOL:=FALSE;
	iStepOsc:INT:=0;
	iOscCounter:INT:=0;
	iStepResetFB:INT:=0;
	dwOldOverride:DWORD:=100;
	lrOverrideVel:LREAL;
(* timer *)
	TimerOutSendPara:TON;
	TimerFileLocked:TON;
(* trigger *)
	RisingEdgeResetFB:R_TRIG;
	RisingEdgeExecute:R_TRIG;
	RisingEdgePowerOn:R_TRIG;
	RisingEdgePowerOff:R_TRIG;
(* Temp variable *)
	xTmp:BOOL:=FALSE;
	wTmp:WORD:=0;
	dwTmp:DWORD:=0;
	dwAdrVar:DWORD:=0;
	rTmpFrequence:REAL;
	lrTmpVelocity:LREAL;
	TimerCommTimeLeft:TON;
	xStartTimerComm:BOOL:=FALSE;
	tTimeCommLeft:TIME;
	TimerCommTimeLeft1:TON;
	xStartTimerComm1:BOOL:=FALSE;
	tTimeCommLeft1:TIME;
	xMovement: BOOL;
	xNoHWError: BOOL;
	iStepCalcRefIndex: INT;
	xCheckRefState: BOOL;
	iTmpFctNr: INT;
	lrTechUnitPerMotorTurn: LREAL;	(* Gilt nur für das Aufsuchen des Reference Index-->Die Technische Einheit muss angegeben werden, damit eine Motorrotation durchgeführt werden kann z.B. 2.5mm/U_Motor  oder 30Grad/U_Motor*)
	xSendBlock: BOOL;
	lrCapturePosition: LREAL;
	xTmpCheckDirectionPos: BOOL;
	xTmpCheckDirectionNeg: BOOL;
	TONWaitCheckHWLimitSwitch: TON;
	xActiveFollowError: BOOL;
	xSetSWPosLimitSwitch: BOOL;
	xResetSWPosLimitSwitch: BOOL;
	iStepSWLimitSwitch: INT;
	lrData: LREAL;
	fbSoEReset: FB_SoEReset;
	xResetAX5000Axis: BOOL;
	iStepResetAX5000FB: INT;
	xTmpHWLimitPos: BOOL;
	xTmpHWLimitNeg: BOOL;
	lrSetPosition: LREAL;
	diStepErrorCounter: DINT;
	diStepErrorCounter1: DINT;
	lrDistance: LREAL;
	xStopAxisVelCtrlActive: BOOL;
	iStopAxis: INT;
	TONWaitStop: TON;
END_VAR
(* Test Timer PUM *)
TimerCommTimeLeft(IN:=xStartTimerComm,PT:=T#99999s);
TimerCommTimeLeft1(IN:=xStartTimerComm1,PT:=T#99999s);
(* reset block function *)
	RisingEdgeResetFB(CLK:=T_Axis.T_CtrleSingle.xReset);
	IF RisingEdgeResetFB.Q THEN
	(* Init. block function *)
		fbAxisReset(Execute:=FALSE, Axis:=T_AxisRefIn);
		fbSoEReset(	sNetId:='' ,bExecute:= FALSE, tTimeout:= T#10s, Axis:= T_AxisRefIn);
		fbAxisPower(	Enable:=FALSE,
					AxisRefIn:=T_AxisRefIn,
					AxisRefOut:=T_AxisRefOut);
		fbAxisStop(Execute:=FALSE, Axis:=T_AxisRefIn);
		fbAxisMoveVelocity(Execute:=FALSE, Axis:=T_AxisRefIn);
		fbAxisMoveAbsolute(Execute:=FALSE, Axis:=T_AxisRefIn);
		fbAxisMoveModulo(Execute:=FALSE, Axis:=T_AxisRefIn);
		fbAxisMoveRelative(Execute:=FALSE, Axis:=T_AxisRefIn);
		fbAxisHoming(	Execute:=FALSE,
						Axis:=T_AxisRefIn,
						AxisOut:=T_AxisRefOut);
		fbAxisSetOverride(Execute:=FALSE,
						AxisRefIn:=T_AxisRefIn,
						AxisRefOut:=T_AxisRefOut);
		fbAxisSetPosition(	Execute:=FALSE, Axis:=T_AxisRefIn);
		fbAxisNewPosAndVel(	Execute:=FALSE,
							Axis:=T_AxisRefIn);
		fbAdsWrite(WRITE:=FALSE);
		fbADS_ReadWriteString(WRTRD:=FALSE);
	(* timer *)
		TimerOutSendPara(IN:=TRUE,PT:=T#1ms);
	(* Init. variable *)
		xResetAxis:=FALSE;
		xResetAX5000Axis:=FALSE;
		xPowerOn:=FALSE;
		xPowerOff:=FALSE;
		xStop:=FALSE;
		xMoveVel:=FALSE;
		iDirectionVel:=1;
		rVelocity:=0;
		xMoveAbs:=FALSE;
		xMoveRel:=FALSE;
		xMoveModulo:=FALSE;
		xHoming:=FALSE;
		xOverride:=FALSE;
		xSetPosition:=FALSE;
		xNewVelocity:=FALSE;
		xNewPosition:=FALSE;
		xCalcAngleRefIndex:=FALSE;
		xSetReferenceFlag:=FALSE;
		xResetReferenceFlag:=FALSE;
		xDefaultAxisParameter:=FALSE;
		xSendAxisParameter:=FALSE;
		xSetSWPosLimitSwitch:=FALSE;
		xResetSWPosLimitSwitch:=FALSE;
		iPtrAxisParameter:=1;
		xSendAxisString:=FALSE;
		iStepSendPara:=0;
		iStepSWLimitSwitch:=0;
		xRestoreAxisPower:=FALSE;
		iStepFile:=0;
		xCtrlePositionOn:=FALSE;
		xCtrlePositionOff:=FALSE;
		xOscillation:=FALSE;
		iStepOsc:=0;
		iOscCounter:=0;
		iStepCalcRefIndex:=0;
	(* int. structure *)
		T_Axis.T_CtrleSingle.dwOverride:=100;
		T_Axis.T_CtrleSingle.iFunction:=0;
		T_Axis.T_CtrleSingle.xDone:=FALSE;
		T_Axis.T_CtrleSingle.xErr:=FALSE;
		T_Axis.T_CtrleSingle.udiErrorID:=0;
		T_Axis.T_CtrleSingle.xPower:=FALSE;
		T_Axis.T_CtrleSingle.xReady:=FALSE;
(*		T_Axis.T_CtrleSingle.xRef:=FALSE;*)
		T_Axis.T_CtrleSingle.xSlave:=FALSE;
		T_Axis.T_CtrleSingle.xConstantVel:=FALSE;
		T_Axis.T_CtrleSingle.xBusyNewPosAndVel:=FALSE;
		T_Axis.T_CtrleSingle.xDriveTorque:=FALSE;
		T_Axis.T_CtrleSingle.xAxisCollisionError:=FALSE;
		(* set flag done *)
		xConfirmResetFB:=TRUE;
		(* disable status flag *)
		T_Axis.T_CtrleSingle.xDone:=FALSE;
		T_Axis.T_CtrleSingle.xErr:=FALSE;
		T_Axis.T_CtrleSingle.udiErrorID:=0;
		(* exit function bloc *)
		(* Test Timer PUM *)
		xStartTimerComm:=FALSE;
		xStartTimerComm1:=FALSE;
		xActiveFollowError:=FALSE;
		IF (T_Axis.T_Config_Gen.iTyp = 1) THEN
			gxZFollowDistanceError:=FALSE;
		END_IF;
		RETURN;
	ELSE
		IF xConfirmResetFB THEN
		(* confirm reset FB *)
			T_Axis.T_CtrleSingle.xDone:=TRUE;
			T_Axis.T_CtrleSingle.xErr:=FALSE;
			T_Axis.T_CtrleSingle.udiErrorID:=0;
			(* reset variable *)
			xConfirmResetFB:=FALSE;
		END_IF
	END_IF

(* return axis state *)
	T_Axis.T_CtrleSingle.xReady:=GETBIT32(T_AxisRefIn.nStateDWord,0) OR gxHardwareOFF;
	IF T_Axis.T_Config_Setting.xAbsoluteEncoder THEN
		T_Axis.T_CtrleSingle.xRef:=xRefHoming;
	ELSE
		T_Axis.T_CtrleSingle.xRef:=GETBIT32(T_AxisRefIn.nStateDWord,1);
	END_IF;
	T_Axis.T_CtrleSingle.xHomingSensor:=xRefHoming;
	T_Axis.T_CtrleSingle.xNotMoving:=GETBIT32(T_AxisRefIn.nStateDWord,2) OR gxHardwareOFF;
	T_Axis.T_CtrleSingle.xSlave:=GETBIT32(T_AxisRefIn.nStateDWord,5);
	T_Axis.T_CtrleSingle.xMovingForward:=GETBIT32(T_AxisRefIn.nStateDWord,9);
	T_Axis.T_CtrleSingle.xMovingBackwards:=GETBIT32(T_AxisRefIn.nStateDWord,10);
	T_Axis.T_CtrleSingle.xConstantVel:=GETBIT32(T_AxisRefIn.nStateDWord,12);
	T_Axis.T_CtrleSingle.xSpindleBlocked:=NOT(T_Axis.T_CtrleSingle.xNotMoving) AND (ABS(T_Axis.T_LiveValue.lrActualVelocity) = 0);
	T_Axis.T_CtrleSingle.xSWLimitSwitchPosActivated:=IxSoftLimitMaxMonitoring;
	IF GETBIT32(T_AxisRefIn.nStateDWord,31) THEN
	(* error servo *)
		T_Axis.T_CtrleSingle.xDone:=FALSE;
		T_Axis.T_CtrleSingle.xErr:=TRUE;
		T_Axis.T_CtrleSingle.udiErrorID:=T_AxisRefIn.nErrorCode;
	END_IF
	(* das Aktivieren dieser Funktion ermöglicht es vom HW Endschalter mittels der Steuerung wegzufahren *)
	T_AxisRefOut.nDeCtrlDWord:=AxisSetAcceptBlockedDriveSignal(nDeCtrlDWord:=T_AxisRefOut.nDeCtrlDWord, bEnable:=T_Axis.T_CtrleSingle.xMoveAwayFromHWLimitSwitchActive);

(* Timer *)
	TimerOutSendPara(IN:=TRUE, PT:=T#10S);
	TimerFileLocked(IN:=TRUE, PT:=T#10S);

(* detection software limit *)
	(* positiv limit *)
	IF T_Axis.T_Config_Setting.xSoftwareLimitPos THEN
		IF AxisSoftLimitMaxExceeded(nStateDWord:=T_AxisRefIn.nStateDWord) THEN
			T_Axis.T_CtrleSingle.xSWLimitPos:=TRUE;
		ELSE
			T_Axis.T_CtrleSingle.xSWLimitPos:=FALSE;
		END_IF;
		T_Axis.T_CtrleSingle.xStateSWLimitPos:=T_Axis.T_CtrleSingle.xSWLimitPos;
	END_IF;
	IF T_Axis.T_Config_Setting.xSoftwareLimitNeg THEN
		IF AxisSoftLimitMinExceeded(nStateDWord:=T_AxisRefIn.nStateDWord) THEN
			T_Axis.T_CtrleSingle.xSWLimitNeg:=TRUE;
		ELSE
			T_Axis.T_CtrleSingle.xSWLimitNeg:=FALSE;
		END_IF;
		T_Axis.T_CtrleSingle.xStateSWLimitNeg:=T_Axis.T_CtrleSingle.xSWLimitNeg;
	END_IF;

(* detection hardware limit *)
	(* positiv limit *)
	IF NOT(T_Axis.T_CtrleSingle.xAX5000Active) THEN
		IF NOT(T_Axis.T_CtrleSingle.xKL2541Active) THEN
			xTmpHWLimitPos:=((USINT_TO_WORD(T_Axis.T_DriveState.usiDriveState1) AND 16#2) = 16#2);
			xTmpHWLimitNeg:=((USINT_TO_WORD(T_Axis.T_DriveState.usiDriveState1) AND 16#4) = 16#4);
		ELSE
			xTmpHWLimitPos:=((UINT_TO_WORD(uiStateAxisZ2_KL2541) AND 16#2) = 16#2);
			xTmpHWLimitNeg:=((UINT_TO_WORD(uiStateAxisZ2_KL2541) AND 16#1) = 16#1);
		END_IF;
	ELSE
		xTmpHWLimitPos:=NOT((wInputState AND wPosLimitSwitchBit) = wPosLimitSwitchBit);
		xTmpHWLimitNeg:=NOT((wInputState AND wNegLimitSwitchBit) = wNegLimitSwitchBit);
	END_IF;
	IF T_Axis.T_Config_Setting.xHardwareLimitPos THEN T_Axis.T_CtrleSingle.xHWLimitPos:=xTmpHWLimitPos;
	ELSE T_Axis.T_CtrleSingle.xHWLimitPos:=FALSE; END_IF
	T_Axis.T_CtrleSingle.xStateHWLimitPos:=T_Axis.T_CtrleSingle.xHWLimitPos;
	(* negativ limit *)
	IF T_Axis.T_Config_Setting.xHardwareLimitNeg THEN T_Axis.T_CtrleSingle.xHWLimitNeg:=xTmpHWLimitNeg;
	ELSE T_Axis.T_CtrleSingle.xHWLimitNeg:=FALSE; END_IF
	T_Axis.T_CtrleSingle.xStateHWLimitNeg:=T_Axis.T_CtrleSingle.xHWLimitNeg;
	xTmpCheckDirectionPos:=	((xMoveVel AND (T_Axis.T_CtrleSingle.lrVelocity >= 0.0)) OR
							(NOT(T_Axis.T_CtrleSingle.xNotMoving) AND (T_Axis.T_CtrleSingle.lrVelocity >= 0.0) AND NOT(xMoveVel) AND NOT(xMoveAbs) AND NOT(xMoveRel)) OR
							(xMoveAbs AND ((T_Axis.T_CtrleSingle.lrPosition - T_Axis.T_LiveValue.lrActualPosition) >= 0)) OR
							(xMoveRel AND (T_Axis.T_CtrleSingle.lrDistance >= 0.0))) AND
							(T_Axis.T_CtrleSingle.xHWLimitPos OR T_Axis.T_CtrleSingle.xSWLimitPos) AND NOT(xHoming);
	xTmpCheckDirectionNeg:=	((xMoveVel AND (T_Axis.T_CtrleSingle.lrVelocity < 0.0)) OR
							(NOT(T_Axis.T_CtrleSingle.xNotMoving) AND (T_Axis.T_CtrleSingle.lrVelocity < 0.0) AND NOT(xMoveVel) AND NOT(xMoveAbs) AND NOT(xMoveRel)) OR
							(xMoveAbs AND ((T_Axis.T_CtrleSingle.lrPosition - T_Axis.T_LiveValue.lrActualPosition) < 0)) OR
							(xMoveRel AND (T_Axis.T_CtrleSingle.lrDistance < 0.0))) AND
							(T_Axis.T_CtrleSingle.xHWLimitNeg OR T_Axis.T_CtrleSingle.xSWLimitNeg) AND NOT(xHoming);
	T_Axis.T_CtrleSingle.xHWLimitPos:=T_Axis.T_CtrleSingle.xHWLimitPos AND xTmpCheckDirectionPos;
	T_Axis.T_CtrleSingle.xHWLimitNeg:=T_Axis.T_CtrleSingle.xHWLimitNeg AND xTmpCheckDirectionNeg;
	T_Axis.T_CtrleSingle.xSWLimitPos:=T_Axis.T_CtrleSingle.xSWLimitPos AND xTmpCheckDirectionPos;
	T_Axis.T_CtrleSingle.xSWLimitNeg:=T_Axis.T_CtrleSingle.xSWLimitNeg AND xTmpCheckDirectionNeg;
	(* monitor hardware limit *)
	IF NOT(T_Axis.T_CtrleSingle.xNotMoving) THEN
		IF T_Axis.T_CtrleSingle.xHWLimitPos OR T_Axis.T_CtrleSingle.xHWLimitNeg OR T_Axis.T_CtrleSingle.xSWLimitPos OR T_Axis.T_CtrleSingle.xSWLimitNeg THEN
		(* set decceleration ramp and make a stop *)
			IF NOT(xStop) THEN
				xStop:=TRUE;
				IF T_Axis.T_CtrleSingle.xHWLimitPos OR T_Axis.T_CtrleSingle.xHWLimitNeg THEN
					xActiveFollowError:=TRUE;
				END_IF;
				IF T_Axis.T_Config_Setting.lrHWLimitDecceleration <> 0 THEN
					T_Axis.T_CtrleSingle.lrDecceleration:=T_Axis.T_Config_Setting.lrHWLimitDecceleration;
				END_IF
			END_IF;
		END_IF
	END_IF
	IF T_Axis.T_CtrleSingle.xNotMoving AND (T_Axis.T_CtrleSingle.xHWLimitPos OR T_Axis.T_CtrleSingle.xHWLimitNeg OR T_Axis.T_CtrleSingle.xSWLimitPos OR T_Axis.T_CtrleSingle.xSWLimitNeg) THEN
		TONWaitCheckHWLimitSwitch(IN:=TRUE,PT:=T#500ms);
		IF TONWaitCheckHWLimitSwitch.Q AND NOT(xStop) THEN
			TONWaitCheckHWLimitSwitch(IN:=FALSE);
			xStop:=TRUE;
			IF T_Axis.T_Config_Setting.lrHWLimitDecceleration <> 0 THEN
				T_Axis.T_CtrleSingle.lrDecceleration:=T_Axis.T_Config_Setting.lrHWLimitDecceleration;
			END_IF
		END_IF;
		IF TONWaitCheckHWLimitSwitch.Q AND xStop THEN
			TONWaitCheckHWLimitSwitch(IN:=FALSE);
		END_IF;
	ELSE
		TONWaitCheckHWLimitSwitch(IN:=FALSE);
	END_IF;

(* detection start *)
	RisingEdgeExecute(CLK:=T_Axis.T_CtrleSingle.xExecute);
	IF RisingEdgeExecute.Q THEN
		RisingEdgeExecute(CLK:=FALSE);
		IF xStop AND (T_Axis.T_CtrleSingle.iFunction <> 1) AND (T_Axis.T_CtrleSingle.iFunction <> 5) AND (T_Axis.T_CtrleSingle.iFunction <> 27) THEN
		(* can not execute a function when 'Stop' activ, except 'Reset' *)
			T_Axis.T_CtrleSingle.xDone:=FALSE;
			T_Axis.T_CtrleSingle.xErr:=TRUE;
			T_Axis.T_CtrleSingle.udiErrorID:=16#F100;		(* Achsfunktion nicht ausführbar wenn Stop-Funktion Aktiv *)
			RETURN;
		END_IF
		CASE T_Axis.T_CtrleSingle.iFunction OF
		(* Reset *)
		1:	xResetAxis:=TRUE;
			iStepResetFB:=1;
			iTmpFctNr:=1;
		(* Power ON *)
		3:	IF NOT(xPowerOn) THEN
				xPowerOn:=TRUE;
				xPowerOff:=NOT(xPowerOn);
				iTmpFctNr:=3;
			ELSE
				T_Axis.T_CtrleSingle.xDone:=TRUE;
				T_Axis.T_CtrleSingle.xErr:= FALSE;
				T_Axis.T_CtrleSingle.udiErrorID:=16#0;
				iTmpFctNr:=3;
				RETURN;
			END_IF;
		(* Power Off *)
		4:	IF xPowerOn THEN
				xPowerOff:=TRUE;
				xPowerOn:=NOT(xPowerOff);
				iTmpFctNr:=4;
			ELSE
				T_Axis.T_CtrleSingle.xDone:=TRUE;
				T_Axis.T_CtrleSingle.xErr:= FALSE;
				T_Axis.T_CtrleSingle.udiErrorID:=16#0;
				iTmpFctNr:=4;
				RETURN;
			END_IF;
		(* Stop *)
		5: 	xStop:=TRUE;
			fbAxisStop(Execute:=FALSE, Axis:=T_AxisRefIn);
			xStartTimerComm1:=TRUE;
			iTmpFctNr:=5;
		(* Velocity *)
		6:	xMoveVel:=TRUE;
			iTmpFctNr:=6;
		(* Absolute *)
		7:	xMoveAbs:=TRUE;
			iTmpFctNr:=7;
		(* Relative *)
		8:	xMoveRel:=TRUE;
			iTmpFctNr:=8;
		(* homing *)
		9:	xHoming:=TRUE;
			iTmpFctNr:=9;
		(* override *)
		10:	xOverride:=TRUE;
			iTmpFctNr:=10;
		(* set position *)
		11:	xSetPosition:=TRUE;
			iTmpFctNr:=11;
		(* change current speed *)
		12:	xNewVelocity:=TRUE;
			T_Axis.T_CtrleSingle.xBusyNewPosAndVel:=TRUE;
			IF xMoveAbs OR xMoveRel OR xMoveModulo OR xOscillation THEN	(* Muss unterschieden werden können, ob Positionsfahrt oder Velocitymode ausgeführt wird *)
				xMovement:=TRUE;
			ELSE
				xMovement:=FALSE;
			END_IF;
			xStartTimerComm:=TRUE;
		(* Set reference flag *)
		13:	xSetReferenceFlag:=TRUE;
			iTmpFctNr:=13;
		(* reset reference flag *)
		14:	xResetReferenceFlag:=TRUE;
			iTmpFctNr:=14;
		(* control position On *)
		15:	xCtrlePositionOn:=TRUE;
			iTmpFctNr:=15;
		(* control position off *)
		16:	xCtrlePositionOff:=TRUE;
			iTmpFctNr:=16;
		(* oscillation *)
		17:	xOscillation:=TRUE;
			iTmpFctNr:=17;
		(* change position *)
		18:	xNewPosition:=TRUE;
			T_Axis.T_CtrleSingle.xBusyNewPosAndVel:=TRUE;
		(* calcultate angle between Reference Index and Reference Sensor *)
		19:	xCalcAngleRefIndex:=TRUE;
			iTmpFctNr:=19;
		(* Default parameter value *)
		20:	xDefaultAxisParameter:=TRUE;
			iTmpFctNr:=20;
		(* Send Parameter *)
		21: 	xSendAxisParameter:=TRUE;
			iPtrAxisParameter:=1;
			iStepSendPara:=1;
			(* copy parameter value *)
			fbDefaultAxisPara(xDefaultValue:=FALSE,T_Axis:=T_Axis);
			iTmpFctNr:=21;
		(* send string *)
		22: 	xSendAxisString:=TRUE;
			sSendAxis:='';
			sReturnAxis:='';
			iTmpFctNr:=22;
		(* Move Modulo *)
		24:	xMoveModulo:=TRUE;
			iTmpFctNr:=24;
		(* Set SW Pos limit switch *)
		25:	xSetSWPosLimitSwitch:=TRUE;
			iStepSWLimitSwitch:=1;
			iTmpFctNr:=25;
		(* Reset SW Pos limit switch *)
		26:	xResetSWPosLimitSwitch:=TRUE;
			iStepSWLimitSwitch:=1;
			iTmpFctNr:=26;
		(* Reset AX5000 Servo function *)
		27:	xResetAX5000Axis:=TRUE;
			iStepResetAX5000FB:=1;
			iTmpFctNr:=27;
		ELSE
		(* function not implemented *)
			T_Axis.T_CtrleSingle.xDone:=FALSE;
			T_Axis.T_CtrleSingle.xErr:=TRUE;
			T_Axis.T_CtrleSingle.udiErrorID:=16#F000;		(* Aufgerufene Achsfunktion besteht nicht *)
			(* Exit FB *)
			RETURN;
		END_CASE
		(* Init. variable *)
		T_Axis.T_CtrleSingle.xDone:=FALSE;
		T_Axis.T_CtrleSingle.xErr:=FALSE;
		T_Axis.T_CtrleSingle.udiErrorID:=0;
		iStopAxis:=1;
		xStopAxisVelCtrlActive:=FALSE;
		IF NOT(xStop) THEN
			T_Axis.T_CtrleSingle.xAxisCollisionError:=FALSE;
		END_IF;
		(* init variable *)
		dwOldOverride:=16#FFFF;
		(* Exit FB *)
		RETURN;
	END_IF

(* Override *)
	IF dwOldOverride <>T_Axis.T_CtrleSingle.dwOverride THEN
		lrOverrideVel:=T_Axis.T_CtrleSingle.lrVelocity; (* T_Axis.T_CtrleSingle.dwOverride / 100;*)
		(* confirm velocity setting *)
		dwOldOverride:=T_Axis.T_CtrleSingle.dwOverride;
	END_IF

(* Reset function *)
	IF xResetAxis THEN
		CASE iStepResetFB OF
		(* check state *)
		1:	xRestoreAxisPower:=FALSE;
			IF xPowerOn THEN iStepResetFB:=10; ELSE iStepResetFB:=20; END_IF
			xActiveFollowError:=FALSE;
			IF (T_Axis.T_Config_Gen.iTyp = 1) THEN
				gxZFollowDistanceError:=FALSE;
			END_IF;
		(* power off *)
		10:	xPowerOff:=TRUE;
			xPowerOn:=NOT(xPowerOff);
			xRestoreAxisPower:=TRUE;
			(* next step *)
			iStepResetFB:=20;
		(* wait power off flag *)
		20:	IF NOT(T_Axis.T_CtrleSingle.xPower) THEN
				fbAxisReset(Execute:=TRUE, Axis:=T_AxisRefIn);
				IF fbAxisReset.Done OR fbAxisReset.Error THEN
					 IF fbAxisReset.Error THEN
						T_Axis.T_CtrleSingle.xDone:=fbAxisReset.Done;
						T_Axis.T_CtrleSingle.xErr:= fbAxisReset.Error;
						T_Axis.T_CtrleSingle.udiErrorID:=fbAxisReset.ErrorID;
					ELSE
					(* activ stop *)
						xStop:=TRUE;
						(* flag reset off only if the power has not to be recovered *)
						IF NOT(xRestoreAxisPower) THEN xResetAxis:=FALSE; END_IF
					END_IF
					(* reset flag busy *)
					T_Axis.T_CtrleSingle.xBusyNewPosAndVel:=FALSE;
					(* init. FB reset *)
					fbAxisReset(Execute:=FALSE, Axis:=T_AxisRefIn);
					(* next step *)
					iStepResetFB:=30;
				END_IF
			END_IF
		(* wait stop done *)
		30:	IF NOT(xStop) OR xStopAxisVelCtrlActive THEN iStepResetFB:=40; END_IF
		(* set power on *)
		40:	xPowerOff:=FALSE;
			xPowerOn:=NOT(xPowerOff);
			(* next step *)
			iStepResetFB:=50;
		(* wait power on flag *)
		50:	IF T_Axis.T_CtrleSingle.xPower THEN
			(* confirm reset *)
				IF NOT(xStopAxisVelCtrlActive) THEN
					T_Axis.T_CtrleSingle.xDone:=TRUE;
					T_Axis.T_CtrleSingle.xErr:= FALSE;
					T_Axis.T_CtrleSingle.udiErrorID:=16#0;
				END_IF;
				(* init. variable *)
				xResetAxis:=FALSE;
			END_IF
		END_CASE
	ELSE fbAxisReset(Execute:=FALSE, Axis:=T_AxisRefIn); END_IF

(* Reset AX5000 Servo function *)
	IF xResetAX5000Axis THEN
		CASE iStepResetAX5000FB OF
		(* check state *)
		1:	xRestoreAxisPower:=FALSE;
			IF xPowerOn THEN iStepResetAX5000FB:=10; ELSE iStepResetAX5000FB:=20; END_IF
			xActiveFollowError:=FALSE;
		(* power off *)
		10:	xPowerOff:=TRUE;
			xPowerOn:=NOT(xPowerOff);
			xRestoreAxisPower:=TRUE;
			(* next step *)
			iStepResetAX5000FB:=20;
		(* wait power off flag *)
		20:	IF NOT(T_Axis.T_CtrleSingle.xPower) THEN
				fbSoEReset(	sNetId:='' ,bExecute:= TRUE, tTimeout:= T#10s, Axis:= T_AxisRefIn);
				IF NOT(fbSoEReset.bBusy) OR fbSoEReset.bError THEN
					 IF fbSoEReset.bError THEN
						T_Axis.T_CtrleSingle.xDone:=NOT(fbSoEReset.bError);
						T_Axis.T_CtrleSingle.xErr:= fbSoEReset.bError;
						IF (fbSoEReset.iSercosErrId <> 0) THEN
							T_Axis.T_CtrleSingle.udiErrorID:=fbSoEReset.iSercosErrId;
						ELSE
							T_Axis.T_CtrleSingle.udiErrorID:=fbSoEReset.iAdsErrId;
						END_IF;
					ELSE
					(* activ stop *)
						xStop:=TRUE;
						(* flag reset off only if the power has not to be recovered *)
						IF NOT(xRestoreAxisPower) THEN
							xResetAX5000Axis:=FALSE;
							T_Axis.T_CtrleSingle.xDone:=TRUE;
							T_Axis.T_CtrleSingle.xErr:= FALSE;
							T_Axis.T_CtrleSingle.udiErrorID:=16#0;
						END_IF
					END_IF
					(* reset flag busy *)
					T_Axis.T_CtrleSingle.xBusyNewPosAndVel:=FALSE;
					(* init. FB reset *)
					fbSoEReset(	sNetId:='' ,bExecute:= FALSE, tTimeout:= T#10s, Axis:= T_AxisRefIn);
					(* next step *)
					iStepResetAX5000FB:=30;
				END_IF
			END_IF
		(* wait stop done *)
		30:	IF NOT(xStop) THEN iStepResetAX5000FB:=40; END_IF
		(* set power on *)
		40:	xPowerOff:=FALSE;
			xPowerOn:=NOT(xPowerOff);
			(* next step *)
			iStepResetAX5000FB:=50;
		(* wait power on flag *)
		50:	IF T_Axis.T_CtrleSingle.xPower THEN
			(* confirm reset *)
				T_Axis.T_CtrleSingle.xDone:=TRUE;
				T_Axis.T_CtrleSingle.xErr:= FALSE;
				T_Axis.T_CtrleSingle.udiErrorID:=16#0;
				(* init. variable *)
				xResetAX5000Axis:=FALSE;
			END_IF
		END_CASE
	ELSE fbSoEReset(	sNetId:='' ,bExecute:= FALSE, tTimeout:= T#10s, Axis:= T_AxisRefIn); END_IF

(* Power function *)
	RisingEdgePowerOn(CLK:=xPowerOn);
	RisingEdgePowerOff(CLK:=xPowerOff);
	IF xPowerOn THEN
		fbAxisPower(	Enable:=TRUE,
					Enable_Positive:=TRUE,
					Enable_Negative:=TRUE,
					Override:= T_Axis.T_CtrleSingle.dwOverride,
					AxisRefIn:=T_AxisRefIn,
					AxisRefOut:=T_AxisRefOut);
		T_Axis.T_CtrleSingle.xPower:=fbAxisPower.Status;
		(* desactiv control flag during sending axis parameter and during reset  *)
		IF NOT(xSendAxisParameter) AND NOT(xResetAxis) AND NOT(xResetAX5000Axis) THEN
			IF RisingEdgePowerOn.Q AND  NOT(fbAxisPower.Error) THEN
				T_Axis.T_CtrleSingle.xDone:=TRUE;
			END_IF
			IF  fbAxisPower.Error THEN
				T_Axis.T_CtrleSingle.xErr:= fbAxisPower.Error;
				T_Axis.T_CtrleSingle.udiErrorID:=fbAxisPower.ErrorID;
			END_IF
		END_IF
	END_IF
	IF xPowerOff THEN
		fbAxisPower(	Enable:=FALSE,
					AxisRefIn:=T_AxisRefIn,
					AxisRefOut:=T_AxisRefOut);
		T_Axis.T_CtrleSingle.xPower:=fbAxisPower.Status;
		(* desactiv control flag during sending axis parameter and during reset *)
		IF NOT(xSendAxisParameter) AND NOT(xResetAxis) AND NOT(xResetAX5000Axis) THEN
			IF RisingEdgePowerOff.Q AND NOT( fbAxisPower.Error) THEN
				T_Axis.T_CtrleSingle.xDone:=TRUE;
			END_IF
			IF  fbAxisPower.Error THEN
				T_Axis.T_CtrleSingle.xErr:= fbAxisPower.Error;
				T_Axis.T_CtrleSingle.udiErrorID:=fbAxisPower.ErrorID;
			END_IF
		END_IF
	END_IF

